ACTION SAW_active:
(*
Copyright (c) 2019 Manuel Goester, Michael Witt, Klaus Kammerer
Institute of Databases and Information Systems, Ulm University, Germany

Permission is hereby granted, free of charge, to any person obtaining a copy 
of this software and associated documentation files (the "Software"), to deal 
in the Software without restriction, including without limitation the rights 
to use, copy, modify, merge, publish, distribute, sublicense, and/or sell 
copies of the Software, and to permit persons to whom the Software is 
furnished to do so, subject to the following conditions:

The above copyright notice and this permission notice shall be included in 
all copies or substantial portions of the Software.

THE SOFTWARE IS PROVIDED "AS IS", WITHOUT WARRANTY OF ANY KIND, EXPRESS OR 
IMPLIED, INCLUDING BUT NOT LIMITED TO THE WARRANTIES OF MERCHANTABILITY, 
FITNESS FOR A PARTICULAR PURPOSE AND NONINFRINGEMENT. IN NO EVENT SHALL THE 
AUTHORS OR COPYRIGHT HOLDERS BE LIABLE FOR ANY CLAIM, DAMAGES OR OTHER 
LIABILITY, WHETHER IN AN ACTION OF CONTRACT, TORT OR OTHERWISE, ARISING FROM, 
OUT OF OR IN CONNECTION WITH THE SOFTWARE OR THE USE OR OTHER DEALINGS 
IN THE SOFTWARE.
*)
CASE stepSaw OF
	1:	
		IF FUR.currWSaw.state <> W_State.NULL THEN
			IF FUR.currWSaw.format.sawEnabled THEN
				// bring w to saw
				//SM.currW.state := StateEnum.AT_FUR_AT_SAW;
				IF NOT(FUR.sRaPosSaw) THEN
					FUR.mRaClockwise := TRUE;
				ELSE
					FUR.mRaClockwise := FALSE;
					stepSaw := stepSaw + 1;
				END_IF
			ELSE
				// skip saw and bring w directly to SL
				stepSaw := stepSaw + 2;
			END_IF
		END_IF
	2:
		// saw
		timer(IN:= TRUE, PT := FUR.currWSaw.format.sawDuration);
		FUR.mSaw := TRUE;
		IF NOT(timer.Q = FALSE AND timer.IN) THEN
			timer(IN:=FALSE);
			FUR.mSaw := FALSE;
			//FUR.state := FUR_State.FUR_SAW_FINISHED;
			stepSaw := stepSaw + 1;
		END_IF
	3: 
		IF SL.currW.state = W_State.NULL THEN
			// bring w to SL
			// SM.currW.state := StateEnum.AT_FUR_ON_CONVEYOR;
			// bend pointers of SL to current workpiece
			SL.bIdx := FUR.bIdxSaw;
			SL.wIdx := FUR.wIdxSaw;
			SL.currW := TC.batchJobQueue.batchJobs[SL.bIdx].workpieces[SL.wIdx];
			// reset own pointers
			FUR.bIdxSaw := 0;
			FUR.wIdxSaw := 0;
			FUR.currWSaw := TC.nullW;
			
			stepSaw := stepSaw + 1;
		ELSE
			// wait for SL to be ready to take a new w
		END_IF
		
	4:
		// bring w to SL
		IF NOT(FUR.sRaPosConveyorBelt) THEN
			FUR.mRaClockwise := TRUE;
		ELSE
			FUR.mRaClockwise := FALSE;
			FUR.compressor := TRUE;
			FUR.valveSlider := TRUE;
		END_IF
		
		IF SL.lbEntry THEN
			FUR.mConveyorBeltForward := TRUE;
		ELSE
			FUR.mConveyorBeltForward := FALSE;
			FUR.compressor := FALSE;
			FUR.valveSlider := FALSE;
			//FUR.state := FUR_State.FUR_W_FINISHED_BACK_TO_DEFAULT;
			stepSaw := stepSaw + 1;
		END_IF
	5:
		// get rotating desk back to succer pos
		IF NOT(FUR.sRaPosSucker) THEN
			FUR.mRaCClockwise := TRUE;
		ELSE
			FUR.mRaCClockwise := FALSE;
			// finsihed, go back to 1 to wait for next w
			stepSaw := 1;
		END_IF
END_CASE
END_ACTION

ACTION TO_DEFAULT_POS_active:
(*
Copyright (c) 2019 Manuel Goester, Michael Witt, Klaus Kammerer
Institute of Databases and Information Systems, Ulm University, Germany

Permission is hereby granted, free of charge, to any person obtaining a copy 
of this software and associated documentation files (the "Software"), to deal 
in the Software without restriction, including without limitation the rights 
to use, copy, modify, merge, publish, distribute, sublicense, and/or sell 
copies of the Software, and to permit persons to whom the Software is 
furnished to do so, subject to the following conditions:

The above copyright notice and this permission notice shall be included in 
all copies or substantial portions of the Software.

THE SOFTWARE IS PROVIDED "AS IS", WITHOUT WARRANTY OF ANY KIND, EXPRESS OR 
IMPLIED, INCLUDING BUT NOT LIMITED TO THE WARRANTIES OF MERCHANTABILITY, 
FITNESS FOR A PARTICULAR PURPOSE AND NONINFRINGEMENT. IN NO EVENT SHALL THE 
AUTHORS OR COPYRIGHT HOLDERS BE LIABLE FOR ANY CLAIM, DAMAGES OR OTHER 
LIABILITY, WHETHER IN AN ACTION OF CONTRACT, TORT OR OTHERWISE, ARISING FROM, 
OUT OF OR IN CONNECTION WITH THE SOFTWARE OR THE USE OR OTHER DEALINGS 
IN THE SOFTWARE.
*)
IF NOT(FUR.sFurnanceSliderOutside) THEN
	FUR.mFurnanceSliderOut := TRUE;
	FUR.compressor := TRUE;
	FUR.valveFurnanceDoor := TRUE;
ELSE
	FUR.mFurnanceSliderOut := FALSE;
	FUR.compressor := FALSE;
	FUR.valveFurnanceDoor := FALSE;
END_IF

IF NOT(FUR.sSuckerPosRa) THEN
	FUR.mSuckertoRa := TRUE;
ELSE
	FUR.mSuckertoRa := FALSE;
END_IF

IF NOT(FUR.sRaPosSucker) THEN
	FUR.mRaCClockwise := TRUE;
ELSE
	FUR.mRaCClockwise := FALSE;
END_IF

IF FUR.sSuckerPosRa AND FUR.sRaPosSucker AND FUR.sFurnanceSliderOutside THEN
	fin := TRUE;
END_IF
END_ACTION

ACTION TO_DEFAULT_POS_exit:
(*
Copyright (c) 2019 Manuel Goester, Michael Witt, Klaus Kammerer
Institute of Databases and Information Systems, Ulm University, Germany

Permission is hereby granted, free of charge, to any person obtaining a copy 
of this software and associated documentation files (the "Software"), to deal 
in the Software without restriction, including without limitation the rights 
to use, copy, modify, merge, publish, distribute, sublicense, and/or sell 
copies of the Software, and to permit persons to whom the Software is 
furnished to do so, subject to the following conditions:

The above copyright notice and this permission notice shall be included in 
all copies or substantial portions of the Software.

THE SOFTWARE IS PROVIDED "AS IS", WITHOUT WARRANTY OF ANY KIND, EXPRESS OR 
IMPLIED, INCLUDING BUT NOT LIMITED TO THE WARRANTIES OF MERCHANTABILITY, 
FITNESS FOR A PARTICULAR PURPOSE AND NONINFRINGEMENT. IN NO EVENT SHALL THE 
AUTHORS OR COPYRIGHT HOLDERS BE LIABLE FOR ANY CLAIM, DAMAGES OR OTHER 
LIABILITY, WHETHER IN AN ACTION OF CONTRACT, TORT OR OTHERWISE, ARISING FROM, 
OUT OF OR IN CONNECTION WITH THE SOFTWARE OR THE USE OR OTHER DEALINGS 
IN THE SOFTWARE.
*)
fin := FALSE;
END_ACTION

END_PROGRAM

// Device/Application/FUR/FBs/FUR_BURN
(*
	Function Block for buring a workpiece in furnace
	w : Workpiece to be burned

Copyright (c) 2019 Manuel Goester, Michael Witt, Klaus Kammerer
Institute of Databases and Information Systems, Ulm University, Germany

Permission is hereby granted, free of charge, to any person obtaining a copy 
of this software and associated documentation files (the "Software"), to deal 
in the Software without restriction, including without limitation the rights 
to use, copy, modify, merge, publish, distribute, sublicense, and/or sell 
copies of the Software, and to permit persons to whom the Software is 
furnished to do so, subject to the following conditions:

The above copyright notice and this permission notice shall be included in 
all copies or substantial portions of the Software.

THE SOFTWARE IS PROVIDED "AS IS", WITHOUT WARRANTY OF ANY KIND, EXPRESS OR 
IMPLIED, INCLUDING BUT NOT LIMITED TO THE WARRANTIES OF MERCHANTABILITY, 
FITNESS FOR A PARTICULAR PURPOSE AND NONINFRINGEMENT. IN NO EVENT SHALL THE 
AUTHORS OR COPYRIGHT HOLDERS BE LIABLE FOR ANY CLAIM, DAMAGES OR OTHER 
LIABILITY, WHETHER IN AN ACTION OF CONTRACT, TORT OR OTHERWISE, ARISING FROM, 
OUT OF OR IN CONNECTION WITH THE SOFTWARE OR THE USE OR OTHER DEALINGS 
IN THE SOFTWARE.
*)
FUNCTION_BLOCK FUR_BURN
VAR_INPUT
	w: Workpiece;
END_VAR
VAR_OUTPUT
END_VAR
VAR
	step: INT := 1;
	fin: BOOL := FALSE;
	stepFin: BOOL := FALSE;
	timer: TON;
END_VAR

CASE step OF
	1:	// open door and drive workpiece into furnace
		// reset flag
		fin := FALSE;
		FUR.compressor := TRUE;
		FUR.valveFurnanceDoor := TRUE;
		IF FUR.sFurnanceSliderInside = FALSE THEN
			FUR.mFurnanceSliderIn := TRUE;
		ELSE
			FUR.mFurnanceSliderIn := FALSE;
			FUR.state := FUR_State.FUR_WAGON_INSIDE;
			step := step + 1;
		END_IF
	2:	// burn
		IF FUR.state = FUR_State.FUR_WAGON_INSIDE THEN
			//SM.currW.state := StateEnum.AT_FUR_IN_FUR;
			timer(IN:= TRUE, PT := FUR.currWBurner.format.furDuration);
			FUR.valveFurnanceDoor := FALSE;
			IF NOT(timer.Q = FALSE AND timer.IN) THEN
				// reset timer
				timer(IN:= FALSE);
				FUR.compressor := TRUE;
				FUR.valveFurnanceDoor := TRUE;
				FUR.state := FUR_State.FUR_BURNED;
				step := step + 1;
			END_IF
		END_IF
	3:	// drive slider out
		IF FUR.state = FUR_State.FUR_BURNED THEN
			//SM.currW.state := StateEnum.AT_FUR_IN_WAGON;
			IF FUR.sFurnanceSliderOutside = FALSE THEN
				FUR.mFurnanceSliderOut := TRUE;
			ELSE
				FUR.mFurnanceSliderOut := FALSE;
				FUR.state := FUR_State.FUR_WAGON_OUTSIDE;
				FUR.compressor := FALSE;
				FUR.valveFurnanceDoor := FALSE;
				step := step + 1;
			END_IF
		END_IF
	4:	// finished
		fin := TRUE;
		step := 1;
END_CASE

END_FUNCTION_BLOCK

// Device/Application/VG/VG_SINGLE_MODE
PROGRAM VG_SINGLE_MODE
VAR
	vg_move: VG_MOVE;
	vg_move_to_pos: VG_MOVE_TO_POS;
	xFin: BOOL;
	yFin: BOOL;
	zFin: BOOL;
	pneumatic_loaded: BOOL;
	timer: TON;
	subBlockStart: BOOL;
	fin: BOOL;
	step: INT := 1;
END_VAR

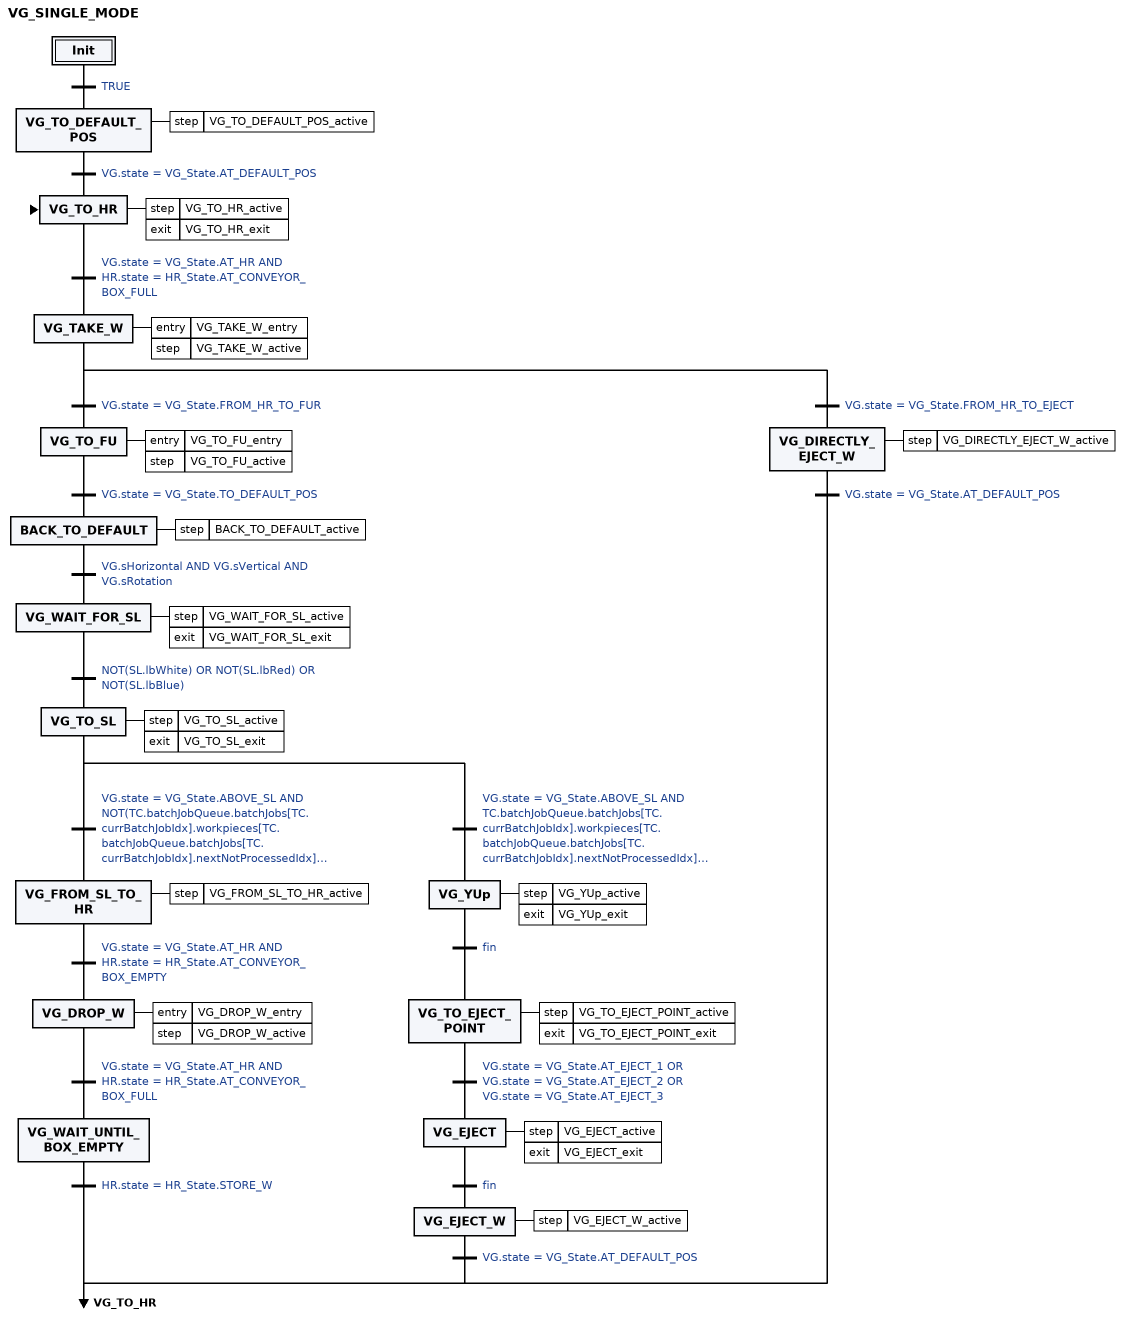
INITIAL_STEP Init:
END_STEP
TRANSITION FROM Init TO VG_TO_DEFAULT_POS
    := TRUE;
END_TRANSITION
STEP VG_TO_DEFAULT_POS:
    VG_TO_DEFAULT_POS_active(N);  // step action
END_STEP
TRANSITION FROM VG_TO_DEFAULT_POS TO VG_TO_HR
    := VG.state = VG_State.AT_DEFAULT_POS;
END_TRANSITION
STEP VG_TO_HR:
    VG_TO_HR_active(N);  // step action
    VG_TO_HR_exit(P0);  // exit action
END_STEP
TRANSITION FROM VG_TO_HR TO VG_TAKE_W
    := VG.state = VG_State.AT_HR AND HR.state = HR_State.AT_CONVEYOR_BOX_FULL;
END_TRANSITION
STEP VG_TAKE_W:
    VG_TAKE_W_entry(P1);  // entry action
    VG_TAKE_W_active(N);  // step action
END_STEP
TRANSITION FROM VG_TAKE_W TO VG_TO_FU
    := VG.state = VG_State.FROM_HR_TO_FUR;
END_TRANSITION
STEP VG_TO_FU:
    VG_TO_FU_entry(P1);  // entry action
    VG_TO_FU_active(N);  // step action
END_STEP
TRANSITION FROM VG_TO_FU TO BACK_TO_DEFAULT
    := VG.state = VG_State.TO_DEFAULT_POS;
END_TRANSITION
STEP BACK_TO_DEFAULT:
    BACK_TO_DEFAULT_active(N);  // step action
END_STEP
TRANSITION FROM BACK_TO_DEFAULT TO VG_WAIT_FOR_SL
    := VG.sHorizontal AND VG.sVertical AND VG.sRotation;
END_TRANSITION
STEP VG_WAIT_FOR_SL:
    VG_WAIT_FOR_SL_active(N);  // step action
    VG_WAIT_FOR_SL_exit(P0);  // exit action
END_STEP
TRANSITION FROM VG_WAIT_FOR_SL TO VG_TO_SL
    := NOT(SL.lbWhite) OR NOT(SL.lbRed) OR NOT(SL.lbBlue);
END_TRANSITION
STEP VG_TO_SL:
    VG_TO_SL_active(N);  // step action
    VG_TO_SL_exit(P0);  // exit action
END_STEP
TRANSITION FROM VG_TO_SL TO VG_FROM_SL_TO_HR
    := VG.state = VG_State.ABOVE_SL AND NOT(TC.batchJobQueue.batchJobs[TC.currBatchJobIdx].workpieces[TC.batchJobQueue.batchJobs[TC.currBatchJobIdx].nextNotProcessedIdx].format.ejectEnabled);
END_TRANSITION
STEP VG_FROM_SL_TO_HR:
    VG_FROM_SL_TO_HR_active(N);  // step action
END_STEP
TRANSITION FROM VG_FROM_SL_TO_HR TO VG_DROP_W
    := VG.state = VG_State.AT_HR AND HR.state = HR_State.AT_CONVEYOR_BOX_EMPTY;
END_TRANSITION
STEP VG_DROP_W:
    VG_DROP_W_entry(P1);  // entry action
    VG_DROP_W_active(N);  // step action
END_STEP
TRANSITION FROM VG_DROP_W TO VG_WAIT_UNTIL_BOX_EMPTY
    := VG.state = VG_State.AT_HR AND HR.state = HR_State.AT_CONVEYOR_BOX_FULL;
END_TRANSITION
STEP VG_WAIT_UNTIL_BOX_EMPTY:
END_STEP
TRANSITION FROM VG_WAIT_UNTIL_BOX_EMPTY TO VG_TO_HR
    := HR.state = HR_State.STORE_W;
END_TRANSITION
TRANSITION FROM VG_TO_SL TO VG_YUp
    := VG.state = VG_State.ABOVE_SL AND TC.batchJobQueue.batchJobs[TC.currBatchJobIdx].workpieces[TC.batchJobQueue.batchJobs[TC.currBatchJobIdx].nextNotProcessedIdx].format.ejectEnabled;
END_TRANSITION
STEP VG_YUp:
    VG_YUp_active(N);  // step action
    VG_YUp_exit(P0);  // exit action
END_STEP
TRANSITION FROM VG_YUp TO VG_TO_EJECT_POINT
    := fin;
END_TRANSITION
STEP VG_TO_EJECT_POINT:
    VG_TO_EJECT_POINT_active(N);  // step action
    VG_TO_EJECT_POINT_exit(P0);  // exit action
END_STEP
TRANSITION FROM VG_TO_EJECT_POINT TO VG_EJECT
    := VG.state = VG_State.AT_EJECT_1 OR VG.state = VG_State.AT_EJECT_2 OR VG.state = VG_State.AT_EJECT_3;
END_TRANSITION
STEP VG_EJECT:
    VG_EJECT_active(N);  // step action
    VG_EJECT_exit(P0);  // exit action
END_STEP
TRANSITION FROM VG_EJECT TO VG_EJECT_W
    := fin;
END_TRANSITION
STEP VG_EJECT_W:
    VG_EJECT_W_active(N);  // step action
END_STEP
TRANSITION FROM VG_EJECT_W TO VG_TO_HR
    := VG.state = VG_State.AT_DEFAULT_POS;
END_TRANSITION
TRANSITION FROM VG_TAKE_W TO VG_DIRECTLY_EJECT_W
    := VG.state = VG_State.FROM_HR_TO_EJECT;
END_TRANSITION
STEP VG_DIRECTLY_EJECT_W:
    VG_DIRECTLY_EJECT_W_active(N);  // step action
END_STEP
TRANSITION FROM VG_DIRECTLY_EJECT_W TO VG_TO_HR
    := VG.state = VG_State.AT_DEFAULT_POS;
END_TRANSITION

ACTION XForward_VG_TAKE_W_active_exit:
(*
Copyright (c) 2019 Manuel Goester, Michael Witt, Klaus Kammerer
Institute of Databases and Information Systems, Ulm University, Germany

Permission is hereby granted, free of charge, to any person obtaining a copy 
of this software and associated documentation files (the "Software"), to deal 
in the Software without restriction, including without limitation the rights 
to use, copy, modify, merge, publish, distribute, sublicense, and/or sell 
copies of the Software, and to permit persons to whom the Software is 
furnished to do so, subject to the following conditions:

The above copyright notice and this permission notice shall be included in 
all copies or substantial portions of the Software.

THE SOFTWARE IS PROVIDED "AS IS", WITHOUT WARRANTY OF ANY KIND, EXPRESS OR 
IMPLIED, INCLUDING BUT NOT LIMITED TO THE WARRANTIES OF MERCHANTABILITY, 
FITNESS FOR A PARTICULAR PURPOSE AND NONINFRINGEMENT. IN NO EVENT SHALL THE 
AUTHORS OR COPYRIGHT HOLDERS BE LIABLE FOR ANY CLAIM, DAMAGES OR OTHER 
LIABILITY, WHETHER IN AN ACTION OF CONTRACT, TORT OR OTHERWISE, ARISING FROM, 
OUT OF OR IN CONNECTION WITH THE SOFTWARE OR THE USE OR OTHER DEALINGS 
IN THE SOFTWARE.
*)
xFin := FALSE;
END_ACTION

ACTION YUp_VG_DROP_W_active_exit:
(*
Copyright (c) 2019 Manuel Goester, Michael Witt, Klaus Kammerer
Institute of Databases and Information Systems, Ulm University, Germany

Permission is hereby granted, free of charge, to any person obtaining a copy 
of this software and associated documentation files (the "Software"), to deal 
in the Software without restriction, including without limitation the rights 
to use, copy, modify, merge, publish, distribute, sublicense, and/or sell 
copies of the Software, and to permit persons to whom the Software is 
furnished to do so, subject to the following conditions:

The above copyright notice and this permission notice shall be included in 
all copies or substantial portions of the Software.

THE SOFTWARE IS PROVIDED "AS IS", WITHOUT WARRANTY OF ANY KIND, EXPRESS OR 
IMPLIED, INCLUDING BUT NOT LIMITED TO THE WARRANTIES OF MERCHANTABILITY, 
FITNESS FOR A PARTICULAR PURPOSE AND NONINFRINGEMENT. IN NO EVENT SHALL THE 
AUTHORS OR COPYRIGHT HOLDERS BE LIABLE FOR ANY CLAIM, DAMAGES OR OTHER 
LIABILITY, WHETHER IN AN ACTION OF CONTRACT, TORT OR OTHERWISE, ARISING FROM, 
OUT OF OR IN CONNECTION WITH THE SOFTWARE OR THE USE OR OTHER DEALINGS 
IN THE SOFTWARE.
*)
yFin := FALSE;
VG.state := VG_State.AT_HR;
VG_SINGLE_MODE.subBlockStart := FALSE;
END_ACTION

ACTION VG_TO_FU_entry:
(*
Copyright (c) 2019 Manuel Goester, Michael Witt, Klaus Kammerer
Institute of Databases and Information Systems, Ulm University, Germany

Permission is hereby granted, free of charge, to any person obtaining a copy 
of this software and associated documentation files (the "Software"), to deal 
in the Software without restriction, including without limitation the rights 
to use, copy, modify, merge, publish, distribute, sublicense, and/or sell 
copies of the Software, and to permit persons to whom the Software is 
furnished to do so, subject to the following conditions:

The above copyright notice and this permission notice shall be included in 
all copies or substantial portions of the Software.

THE SOFTWARE IS PROVIDED "AS IS", WITHOUT WARRANTY OF ANY KIND, EXPRESS OR 
IMPLIED, INCLUDING BUT NOT LIMITED TO THE WARRANTIES OF MERCHANTABILITY, 
FITNESS FOR A PARTICULAR PURPOSE AND NONINFRINGEMENT. IN NO EVENT SHALL THE 
AUTHORS OR COPYRIGHT HOLDERS BE LIABLE FOR ANY CLAIM, DAMAGES OR OTHER 
LIABILITY, WHETHER IN AN ACTION OF CONTRACT, TORT OR OTHERWISE, ARISING FROM, 
OUT OF OR IN CONNECTION WITH THE SOFTWARE OR THE USE OR OTHER DEALINGS 
IN THE SOFTWARE.
*)
VG_SINGLE_MODE.subBlockStart := TRUE;
END_ACTION

ACTION ZBack_VG_FROM_SL_TO_HR_active_exit:
(*
Copyright (c) 2019 Manuel Goester, Michael Witt, Klaus Kammerer
Institute of Databases and Information Systems, Ulm University, Germany

Permission is hereby granted, free of charge, to any person obtaining a copy 
of this software and associated documentation files (the "Software"), to deal 
in the Software without restriction, including without limitation the rights 
to use, copy, modify, merge, publish, distribute, sublicense, and/or sell 
copies of the Software, and to permit persons to whom the Software is 
furnished to do so, subject to the following conditions:

The above copyright notice and this permission notice shall be included in 
all copies or substantial portions of the Software.

THE SOFTWARE IS PROVIDED "AS IS", WITHOUT WARRANTY OF ANY KIND, EXPRESS OR 
IMPLIED, INCLUDING BUT NOT LIMITED TO THE WARRANTIES OF MERCHANTABILITY, 
FITNESS FOR A PARTICULAR PURPOSE AND NONINFRINGEMENT. IN NO EVENT SHALL THE 
AUTHORS OR COPYRIGHT HOLDERS BE LIABLE FOR ANY CLAIM, DAMAGES OR OTHER 
LIABILITY, WHETHER IN AN ACTION OF CONTRACT, TORT OR OTHERWISE, ARISING FROM, 
OUT OF OR IN CONNECTION WITH THE SOFTWARE OR THE USE OR OTHER DEALINGS 
IN THE SOFTWARE.
*)
zFin := FALSE;
END_ACTION

ACTION Suction_VG_TAKE_W_active_active:
(*
Copyright (c) 2019 Manuel Goester, Michael Witt, Klaus Kammerer
Institute of Databases and Information Systems, Ulm University, Germany

Permission is hereby granted, free of charge, to any person obtaining a copy 
of this software and associated documentation files (the "Software"), to deal 
in the Software without restriction, including without limitation the rights 
to use, copy, modify, merge, publish, distribute, sublicense, and/or sell 
copies of the Software, and to permit persons to whom the Software is 
furnished to do so, subject to the following conditions:

The above copyright notice and this permission notice shall be included in 
all copies or substantial portions of the Software.

THE SOFTWARE IS PROVIDED "AS IS", WITHOUT WARRANTY OF ANY KIND, EXPRESS OR 
IMPLIED, INCLUDING BUT NOT LIMITED TO THE WARRANTIES OF MERCHANTABILITY, 
FITNESS FOR A PARTICULAR PURPOSE AND NONINFRINGEMENT. IN NO EVENT SHALL THE 
AUTHORS OR COPYRIGHT HOLDERS BE LIABLE FOR ANY CLAIM, DAMAGES OR OTHER 
LIABILITY, WHETHER IN AN ACTION OF CONTRACT, TORT OR OTHERWISE, ARISING FROM, 
OUT OF OR IN CONNECTION WITH THE SOFTWARE OR THE USE OR OTHER DEALINGS 
IN THE SOFTWARE.
*)
IF pneumatic_loaded = FALSE THEN
	VG.valve := TRUE;
	// init timer
	timer(IN:= TRUE, PT:= T#2S);
	
	IF timer.Q = FALSE AND timer.IN THEN
		// go
		VG.compressor := TRUE;
	ELSE
		// stop
		VG.compressor := FALSE;
		
		// reset timer
		timer(IN:= FALSE);
		
		// go to next step
		pneumatic_loaded := TRUE;
	END_IF
ELSE
	// reset timer
	timer(IN:= FALSE);
END_IF
END_ACTION

ACTION ZBack_VG_TO_FU_active_active:
(*
Copyright (c) 2019 Manuel Goester, Michael Witt, Klaus Kammerer
Institute of Databases and Information Systems, Ulm University, Germany

Permission is hereby granted, free of charge, to any person obtaining a copy 
of this software and associated documentation files (the "Software"), to deal 
in the Software without restriction, including without limitation the rights 
to use, copy, modify, merge, publish, distribute, sublicense, and/or sell 
copies of the Software, and to permit persons to whom the Software is 
furnished to do so, subject to the following conditions:

The above copyright notice and this permission notice shall be included in 
all copies or substantial portions of the Software.

THE SOFTWARE IS PROVIDED "AS IS", WITHOUT WARRANTY OF ANY KIND, EXPRESS OR 
IMPLIED, INCLUDING BUT NOT LIMITED TO THE WARRANTIES OF MERCHANTABILITY, 
FITNESS FOR A PARTICULAR PURPOSE AND NONINFRINGEMENT. IN NO EVENT SHALL THE 
AUTHORS OR COPYRIGHT HOLDERS BE LIABLE FOR ANY CLAIM, DAMAGES OR OTHER 
LIABILITY, WHETHER IN AN ACTION OF CONTRACT, TORT OR OTHERWISE, ARISING FROM, 
OUT OF OR IN CONNECTION WITH THE SOFTWARE OR THE USE OR OTHER DEALINGS 
IN THE SOFTWARE.
*)
IF NOT(VG.sHorizontal) THEN
	VG.mHorizontalBackward := TRUE;
ELSE
	VG.mHorizontalBackward := FALSE;
	zFin := TRUE;
END_IF
END_ACTION

ACTION VG_TO_SL_active:
(*
Copyright (c) 2019 Manuel Goester, Michael Witt, Klaus Kammerer
Institute of Databases and Information Systems, Ulm University, Germany

Permission is hereby granted, free of charge, to any person obtaining a copy 
of this software and associated documentation files (the "Software"), to deal 
in the Software without restriction, including without limitation the rights 
to use, copy, modify, merge, publish, distribute, sublicense, and/or sell 
copies of the Software, and to permit persons to whom the Software is 
furnished to do so, subject to the following conditions:

The above copyright notice and this permission notice shall be included in 
all copies or substantial portions of the Software.

THE SOFTWARE IS PROVIDED "AS IS", WITHOUT WARRANTY OF ANY KIND, EXPRESS OR 
IMPLIED, INCLUDING BUT NOT LIMITED TO THE WARRANTIES OF MERCHANTABILITY, 
FITNESS FOR A PARTICULAR PURPOSE AND NONINFRINGEMENT. IN NO EVENT SHALL THE 
AUTHORS OR COPYRIGHT HOLDERS BE LIABLE FOR ANY CLAIM, DAMAGES OR OTHER 
LIABILITY, WHETHER IN AN ACTION OF CONTRACT, TORT OR OTHERWISE, ARISING FROM, 
OUT OF OR IN CONNECTION WITH THE SOFTWARE OR THE USE OR OTHER DEALINGS 
IN THE SOFTWARE.
*)
CASE step OF
	1:
		// decide to which positon of SL VG will go
		IF NOT(SL.lbWhite) THEN
			// go to sorting line pos 1: 
			VG.state := VG_State.TO_SL_OUTPUT_1;
			step := step + 1;
		ELSIF NOT(SL.lbRed) THEN
			// go to sorting line pos 2: 
			VG.state := VG_State.TO_SL_OUTPUT_2;
			step := step + 1;
		ELSIF NOT(SL.lbBlue) THEN
			// go to sorting line pos 3: 
			VG.state := VG_State.TO_SL_OUTPUT_3;
			step := step + 1;
		END_IF
	2:
		// x and z axis: move to SL 
		IF NOT(fin) THEN
			CASE VG.state OF
				VG_State.TO_SL_OUTPUT_1:
					vg_move_to_pos(x := 58, y := 0, z := 69);
				VG_State.TO_SL_OUTPUT_2:
					vg_move_to_pos(x := 63, y := 0, z := 57);
				VG_State.TO_SL_OUTPUT_3:
					vg_move_to_pos(x := 87, y := 0, z := 47);
			END_CASE
			fin := vg_move_to_pos.fin;
		ELSE
			fin := FALSE;
			step := step + 1;
		END_IF
	3:
		// y axis: move to SL
		IF NOT(fin) THEN
			CASE VG.state OF
				VG_State.TO_SL_OUTPUT_1:
					vg_move_to_pos(x := 58, y := 125, z := 69);
					TC.batchJobQueue.batchJobs[TC.currBatchJobIdx].workpieces[TC.batchJobQueue.batchJobs[TC.currBatchJobIdx].nextNotProcessedIdx].sortingLinePos := 1;
				VG_State.TO_SL_OUTPUT_2:
					vg_move_to_pos(x := 63, y := 125, z := 57);
					TC.batchJobQueue.batchJobs[TC.currBatchJobIdx].workpieces[TC.batchJobQueue.batchJobs[TC.currBatchJobIdx].nextNotProcessedIdx].sortingLinePos := 2;
				VG_State.TO_SL_OUTPUT_3:
					vg_move_to_pos(x := 87, y := 125, z := 47);
					TC.batchJobQueue.batchJobs[TC.currBatchJobIdx].workpieces[TC.batchJobQueue.batchJobs[TC.currBatchJobIdx].nextNotProcessedIdx].sortingLinePos := 3;
			END_CASE
			fin := vg_move_to_pos.fin;
		ELSE
			fin := FALSE;
			step := step + 1;
		END_IF
	4:
		CASE VG.state OF
			VG_State.TO_SL_OUTPUT_1:
				VG.state := VG_State.AT_SL_OUTPUT_1;
			VG_State.TO_SL_OUTPUT_2:
				VG.state := VG_State.AT_SL_OUTPUT_2;
			VG_State.TO_SL_OUTPUT_3:
				VG.state := VG_State.AT_SL_OUTPUT_3;
		END_CASE
		// succ workpiece
		IF pneumatic_loaded = FALSE THEN
			VG.valve := TRUE;
			// init timer
			timer(IN:= TRUE, PT:= T#2S);
			IF timer.Q = FALSE AND timer.IN THEN
				// go
				VG.compressor := TRUE;
			ELSE
				// stop
				VG.compressor := FALSE;
				// reset timer
				timer(IN:= FALSE);
				// set flag
				pneumatic_loaded := TRUE;
			END_IF
		ELSE
			step := step + 1;
		END_IF
	5:
		// y axis: move up
		IF NOT(VG.sVertical) THEN
			VG.mVerticalUp := TRUE;
		ELSE
			VG.mVerticalUp := FALSE;
			VG.cY := 0;
			step := step + 1;
		END_IF
	6:
		// finsihed
		VG.state := VG_State.ABOVE_SL;
END_CASE
END_ACTION

ACTION YDown_VG_TO_FU_active_exit:
(*
Copyright (c) 2019 Manuel Goester, Michael Witt, Klaus Kammerer
Institute of Databases and Information Systems, Ulm University, Germany

Permission is hereby granted, free of charge, to any person obtaining a copy 
of this software and associated documentation files (the "Software"), to deal 
in the Software without restriction, including without limitation the rights 
to use, copy, modify, merge, publish, distribute, sublicense, and/or sell 
copies of the Software, and to permit persons to whom the Software is 
furnished to do so, subject to the following conditions:

The above copyright notice and this permission notice shall be included in 
all copies or substantial portions of the Software.

THE SOFTWARE IS PROVIDED "AS IS", WITHOUT WARRANTY OF ANY KIND, EXPRESS OR 
IMPLIED, INCLUDING BUT NOT LIMITED TO THE WARRANTIES OF MERCHANTABILITY, 
FITNESS FOR A PARTICULAR PURPOSE AND NONINFRINGEMENT. IN NO EVENT SHALL THE 
AUTHORS OR COPYRIGHT HOLDERS BE LIABLE FOR ANY CLAIM, DAMAGES OR OTHER 
LIABILITY, WHETHER IN AN ACTION OF CONTRACT, TORT OR OTHERWISE, ARISING FROM, 
OUT OF OR IN CONNECTION WITH THE SOFTWARE OR THE USE OR OTHER DEALINGS 
IN THE SOFTWARE.
*)
fin := FALSE;
END_ACTION

ACTION ZBack_VG_TO_FU_active_exit_0:
(*
Copyright (c) 2019 Manuel Goester, Michael Witt, Klaus Kammerer
Institute of Databases and Information Systems, Ulm University, Germany

Permission is hereby granted, free of charge, to any person obtaining a copy 
of this software and associated documentation files (the "Software"), to deal 
in the Software without restriction, including without limitation the rights 
to use, copy, modify, merge, publish, distribute, sublicense, and/or sell 
copies of the Software, and to permit persons to whom the Software is 
furnished to do so, subject to the following conditions:

The above copyright notice and this permission notice shall be included in 
all copies or substantial portions of the Software.

THE SOFTWARE IS PROVIDED "AS IS", WITHOUT WARRANTY OF ANY KIND, EXPRESS OR 
IMPLIED, INCLUDING BUT NOT LIMITED TO THE WARRANTIES OF MERCHANTABILITY, 
FITNESS FOR A PARTICULAR PURPOSE AND NONINFRINGEMENT. IN NO EVENT SHALL THE 
AUTHORS OR COPYRIGHT HOLDERS BE LIABLE FOR ANY CLAIM, DAMAGES OR OTHER 
LIABILITY, WHETHER IN AN ACTION OF CONTRACT, TORT OR OTHERWISE, ARISING FROM, 
OUT OF OR IN CONNECTION WITH THE SOFTWARE OR THE USE OR OTHER DEALINGS 
IN THE SOFTWARE.
*)
zFin := FALSE;
END_ACTION

ACTION Wait_VG_DROP_W_active_active:
(*
Copyright (c) 2019 Manuel Goester, Michael Witt, Klaus Kammerer
Institute of Databases and Information Systems, Ulm University, Germany

Permission is hereby granted, free of charge, to any person obtaining a copy 
of this software and associated documentation files (the "Software"), to deal 
in the Software without restriction, including without limitation the rights 
to use, copy, modify, merge, publish, distribute, sublicense, and/or sell 
copies of the Software, and to permit persons to whom the Software is 
furnished to do so, subject to the following conditions:

The above copyright notice and this permission notice shall be included in 
all copies or substantial portions of the Software.

THE SOFTWARE IS PROVIDED "AS IS", WITHOUT WARRANTY OF ANY KIND, EXPRESS OR 
IMPLIED, INCLUDING BUT NOT LIMITED TO THE WARRANTIES OF MERCHANTABILITY, 
FITNESS FOR A PARTICULAR PURPOSE AND NONINFRINGEMENT. IN NO EVENT SHALL THE 
AUTHORS OR COPYRIGHT HOLDERS BE LIABLE FOR ANY CLAIM, DAMAGES OR OTHER 
LIABILITY, WHETHER IN AN ACTION OF CONTRACT, TORT OR OTHERWISE, ARISING FROM, 
OUT OF OR IN CONNECTION WITH THE SOFTWARE OR THE USE OR OTHER DEALINGS 
IN THE SOFTWARE.
*)
timer(IN:= TRUE, PT:= T#1S);
IF NOT(timer.Q = FALSE AND timer.IN) THEN
	// reset timer
	timer(IN:= FALSE);
	// go to next step
	fin := TRUE;
END_IF
END_ACTION

ACTION XForward_VG_TAKE_W_active_active:
(*
Copyright (c) 2019 Manuel Goester, Michael Witt, Klaus Kammerer
Institute of Databases and Information Systems, Ulm University, Germany

Permission is hereby granted, free of charge, to any person obtaining a copy 
of this software and associated documentation files (the "Software"), to deal 
in the Software without restriction, including without limitation the rights 
to use, copy, modify, merge, publish, distribute, sublicense, and/or sell 
copies of the Software, and to permit persons to whom the Software is 
furnished to do so, subject to the following conditions:

The above copyright notice and this permission notice shall be included in 
all copies or substantial portions of the Software.

THE SOFTWARE IS PROVIDED "AS IS", WITHOUT WARRANTY OF ANY KIND, EXPRESS OR 
IMPLIED, INCLUDING BUT NOT LIMITED TO THE WARRANTIES OF MERCHANTABILITY, 
FITNESS FOR A PARTICULAR PURPOSE AND NONINFRINGEMENT. IN NO EVENT SHALL THE 
AUTHORS OR COPYRIGHT HOLDERS BE LIABLE FOR ANY CLAIM, DAMAGES OR OTHER 
LIABILITY, WHETHER IN AN ACTION OF CONTRACT, TORT OR OTHERWISE, ARISING FROM, 
OUT OF OR IN CONNECTION WITH THE SOFTWARE OR THE USE OR OTHER DEALINGS 
IN THE SOFTWARE.
*)
VG.state := VG_State.GET_W_FROM_HR;
IF NOT(xFin) THEN
	vg_move_to_pos(x:=27, y:=0, z:=206);
	xFin := vg_move_to_pos.fin;
END_IF
END_ACTION

ACTION Wait_VG_TO_FU_active_exit:
(*
Copyright (c) 2019 Manuel Goester, Michael Witt, Klaus Kammerer
Institute of Databases and Information Systems, Ulm University, Germany

Permission is hereby granted, free of charge, to any person obtaining a copy 
of this software and associated documentation files (the "Software"), to deal 
in the Software without restriction, including without limitation the rights 
to use, copy, modify, merge, publish, distribute, sublicense, and/or sell 
copies of the Software, and to permit persons to whom the Software is 
furnished to do so, subject to the following conditions:

The above copyright notice and this permission notice shall be included in 
all copies or substantial portions of the Software.

THE SOFTWARE IS PROVIDED "AS IS", WITHOUT WARRANTY OF ANY KIND, EXPRESS OR 
IMPLIED, INCLUDING BUT NOT LIMITED TO THE WARRANTIES OF MERCHANTABILITY, 
FITNESS FOR A PARTICULAR PURPOSE AND NONINFRINGEMENT. IN NO EVENT SHALL THE 
AUTHORS OR COPYRIGHT HOLDERS BE LIABLE FOR ANY CLAIM, DAMAGES OR OTHER 
LIABILITY, WHETHER IN AN ACTION OF CONTRACT, TORT OR OTHERWISE, ARISING FROM, 
OUT OF OR IN CONNECTION WITH THE SOFTWARE OR THE USE OR OTHER DEALINGS 
IN THE SOFTWARE.
*)
fin := FALSE;
END_ACTION

ACTION YDown_VG_DROP_W_active_active:
(*
Copyright (c) 2019 Manuel Goester, Michael Witt, Klaus Kammerer
Institute of Databases and Information Systems, Ulm University, Germany

Permission is hereby granted, free of charge, to any person obtaining a copy 
of this software and associated documentation files (the "Software"), to deal 
in the Software without restriction, including without limitation the rights 
to use, copy, modify, merge, publish, distribute, sublicense, and/or sell 
copies of the Software, and to permit persons to whom the Software is 
furnished to do so, subject to the following conditions:

The above copyright notice and this permission notice shall be included in 
all copies or substantial portions of the Software.

THE SOFTWARE IS PROVIDED "AS IS", WITHOUT WARRANTY OF ANY KIND, EXPRESS OR 
IMPLIED, INCLUDING BUT NOT LIMITED TO THE WARRANTIES OF MERCHANTABILITY, 
FITNESS FOR A PARTICULAR PURPOSE AND NONINFRINGEMENT. IN NO EVENT SHALL THE 
AUTHORS OR COPYRIGHT HOLDERS BE LIABLE FOR ANY CLAIM, DAMAGES OR OTHER 
LIABILITY, WHETHER IN AN ACTION OF CONTRACT, TORT OR OTHERWISE, ARISING FROM, 
OUT OF OR IN CONNECTION WITH THE SOFTWARE OR THE USE OR OTHER DEALINGS 
IN THE SOFTWARE.
*)
VG.state := VG_State.DROPPING_W_TO_HR;
IF NOT(yFin) THEN
	vg_move_to_pos(x:=27, y:=45, z:=206);
	IF vg_move_to_pos.fin THEN
		yFin := TRUE;
	END_IF
END_IF
END_ACTION

ACTION VG_TO_EJECT_POINT_active:
(*
Copyright (c) 2019 Manuel Goester, Michael Witt, Klaus Kammerer
Institute of Databases and Information Systems, Ulm University, Germany

Permission is hereby granted, free of charge, to any person obtaining a copy 
of this software and associated documentation files (the "Software"), to deal 
in the Software without restriction, including without limitation the rights 
to use, copy, modify, merge, publish, distribute, sublicense, and/or sell 
copies of the Software, and to permit persons to whom the Software is 
furnished to do so, subject to the following conditions:

The above copyright notice and this permission notice shall be included in 
all copies or substantial portions of the Software.

THE SOFTWARE IS PROVIDED "AS IS", WITHOUT WARRANTY OF ANY KIND, EXPRESS OR 
IMPLIED, INCLUDING BUT NOT LIMITED TO THE WARRANTIES OF MERCHANTABILITY, 
FITNESS FOR A PARTICULAR PURPOSE AND NONINFRINGEMENT. IN NO EVENT SHALL THE 
AUTHORS OR COPYRIGHT HOLDERS BE LIABLE FOR ANY CLAIM, DAMAGES OR OTHER 
LIABILITY, WHETHER IN AN ACTION OF CONTRACT, TORT OR OTHERWISE, ARISING FROM, 
OUT OF OR IN CONNECTION WITH THE SOFTWARE OR THE USE OR OTHER DEALINGS 
IN THE SOFTWARE.
*)
IF NOT(fin) THEN
	IF TC.batchJobQueue.batchJobs[TC.currBatchJobIdx].workpieces[TC.batchJobQueue.batchJobs[TC.currBatchJobIdx].nextNotProcessedIdx].sortingLinePos = 1 THEN
		// go to eject point 1
		vg_move_to_pos(x := 25, y := 133, z := 2);
	ELSIF TC.batchJobQueue.batchJobs[TC.currBatchJobIdx].workpieces[TC.batchJobQueue.batchJobs[TC.currBatchJobIdx].nextNotProcessedIdx].sortingLinePos = 2 THEN
		// go to eject point 2
		vg_move_to_pos(x := 30, y := 133, z := 15);
	ELSE
		// go to eject point 3
		vg_move_to_pos(x := 49, y := 133, z := 23);
	END_IF
	fin := vg_move_to_pos.fin;
	IF fin THEN
		IF TC.batchJobQueue.batchJobs[TC.currBatchJobIdx].workpieces[TC.batchJobQueue.batchJobs[TC.currBatchJobIdx].nextNotProcessedIdx].sortingLinePos = 1 THEN
			VG.state := VG_State.AT_EJECT_1;
		ELSIF TC.batchJobQueue.batchJobs[TC.currBatchJobIdx].workpieces[TC.batchJobQueue.batchJobs[TC.currBatchJobIdx].nextNotProcessedIdx].sortingLinePos = 2 THEN
			VG.state := VG_State.AT_EJECT_2;
		ELSE
			VG.state := VG_State.AT_EJECT_3;
		END_IF
	END_IF
END_IF
END_ACTION

ACTION YDown_VG_DROP_W_active_exit:
(*
Copyright (c) 2019 Manuel Goester, Michael Witt, Klaus Kammerer
Institute of Databases and Information Systems, Ulm University, Germany

Permission is hereby granted, free of charge, to any person obtaining a copy 
of this software and associated documentation files (the "Software"), to deal 
in the Software without restriction, including without limitation the rights 
to use, copy, modify, merge, publish, distribute, sublicense, and/or sell 
copies of the Software, and to permit persons to whom the Software is 
furnished to do so, subject to the following conditions:

The above copyright notice and this permission notice shall be included in 
all copies or substantial portions of the Software.

THE SOFTWARE IS PROVIDED "AS IS", WITHOUT WARRANTY OF ANY KIND, EXPRESS OR 
IMPLIED, INCLUDING BUT NOT LIMITED TO THE WARRANTIES OF MERCHANTABILITY, 
FITNESS FOR A PARTICULAR PURPOSE AND NONINFRINGEMENT. IN NO EVENT SHALL THE 
AUTHORS OR COPYRIGHT HOLDERS BE LIABLE FOR ANY CLAIM, DAMAGES OR OTHER 
LIABILITY, WHETHER IN AN ACTION OF CONTRACT, TORT OR OTHERWISE, ARISING FROM, 
OUT OF OR IN CONNECTION WITH THE SOFTWARE OR THE USE OR OTHER DEALINGS 
IN THE SOFTWARE.
*)
yFin := FALSE;
END_ACTION

ACTION OpenVentil_VG_DROP_W_active_exit:
(*
Copyright (c) 2019 Manuel Goester, Michael Witt, Klaus Kammerer
Institute of Databases and Information Systems, Ulm University, Germany

Permission is hereby granted, free of charge, to any person obtaining a copy 
of this software and associated documentation files (the "Software"), to deal 
in the Software without restriction, including without limitation the rights 
to use, copy, modify, merge, publish, distribute, sublicense, and/or sell 
copies of the Software, and to permit persons to whom the Software is 
furnished to do so, subject to the following conditions:

The above copyright notice and this permission notice shall be included in 
all copies or substantial portions of the Software.

THE SOFTWARE IS PROVIDED "AS IS", WITHOUT WARRANTY OF ANY KIND, EXPRESS OR 
IMPLIED, INCLUDING BUT NOT LIMITED TO THE WARRANTIES OF MERCHANTABILITY, 
FITNESS FOR A PARTICULAR PURPOSE AND NONINFRINGEMENT. IN NO EVENT SHALL THE 
AUTHORS OR COPYRIGHT HOLDERS BE LIABLE FOR ANY CLAIM, DAMAGES OR OTHER 
LIABILITY, WHETHER IN AN ACTION OF CONTRACT, TORT OR OTHERWISE, ARISING FROM, 
OUT OF OR IN CONNECTION WITH THE SOFTWARE OR THE USE OR OTHER DEALINGS 
IN THE SOFTWARE.
*)
END_ACTION

ACTION VG_EJECT_W_active:
(*
Copyright (c) 2019 Manuel Goester, Michael Witt, Klaus Kammerer
Institute of Databases and Information Systems, Ulm University, Germany

Permission is hereby granted, free of charge, to any person obtaining a copy 
of this software and associated documentation files (the "Software"), to deal 
in the Software without restriction, including without limitation the rights 
to use, copy, modify, merge, publish, distribute, sublicense, and/or sell 
copies of the Software, and to permit persons to whom the Software is 
furnished to do so, subject to the following conditions:

The above copyright notice and this permission notice shall be included in 
all copies or substantial portions of the Software.

THE SOFTWARE IS PROVIDED "AS IS", WITHOUT WARRANTY OF ANY KIND, EXPRESS OR 
IMPLIED, INCLUDING BUT NOT LIMITED TO THE WARRANTIES OF MERCHANTABILITY, 
FITNESS FOR A PARTICULAR PURPOSE AND NONINFRINGEMENT. IN NO EVENT SHALL THE 
AUTHORS OR COPYRIGHT HOLDERS BE LIABLE FOR ANY CLAIM, DAMAGES OR OTHER 
LIABILITY, WHETHER IN AN ACTION OF CONTRACT, TORT OR OTHERWISE, ARISING FROM, 
OUT OF OR IN CONNECTION WITH THE SOFTWARE OR THE USE OR OTHER DEALINGS 
IN THE SOFTWARE.
*)
// Brings VG to its default pos where sVertical = sHorizontal = sRotation = 1
// 1. y-Axis 2. z-Axis 3. rotation
IF NOT(VG.sVertical) THEN
	VG.mVerticalUp := TRUE;
ELSE
	VG.mVerticalUp := FALSE;
	VG.cY := 0;
END_IF
IF NOT(VG.sHorizontal) THEN
	VG.mHorizontalBackward := TRUE;
ELSE
	VG.mHorizontalBackward := FALSE;
	VG.cX := 0;
END_IF
IF NOT(VG.sRotation) THEN
	VG.mRotationClockwise := TRUE;
ELSE
	VG.mRotationClockwise := FALSE;
	VG.cZ := 0;
END_IF

IF VG.sHorizontal AND VG.sVertical AND VG.sRotation THEN
	// default pos reached
	VG.state := VG_State.AT_DEFAULT_POS;
END_IF
END_ACTION

ACTION OpenVentil_VG_DROP_W_active_active:
(*
Copyright (c) 2019 Manuel Goester, Michael Witt, Klaus Kammerer
Institute of Databases and Information Systems, Ulm University, Germany

Permission is hereby granted, free of charge, to any person obtaining a copy 
of this software and associated documentation files (the "Software"), to deal 
in the Software without restriction, including without limitation the rights 
to use, copy, modify, merge, publish, distribute, sublicense, and/or sell 
copies of the Software, and to permit persons to whom the Software is 
furnished to do so, subject to the following conditions:

The above copyright notice and this permission notice shall be included in 
all copies or substantial portions of the Software.

THE SOFTWARE IS PROVIDED "AS IS", WITHOUT WARRANTY OF ANY KIND, EXPRESS OR 
IMPLIED, INCLUDING BUT NOT LIMITED TO THE WARRANTIES OF MERCHANTABILITY, 
FITNESS FOR A PARTICULAR PURPOSE AND NONINFRINGEMENT. IN NO EVENT SHALL THE 
AUTHORS OR COPYRIGHT HOLDERS BE LIABLE FOR ANY CLAIM, DAMAGES OR OTHER 
LIABILITY, WHETHER IN AN ACTION OF CONTRACT, TORT OR OTHERWISE, ARISING FROM, 
OUT OF OR IN CONNECTION WITH THE SOFTWARE OR THE USE OR OTHER DEALINGS 
IN THE SOFTWARE.
*)
VG.valve := FALSE;
pneumatic_loaded := FALSE;
END_ACTION

ACTION ZBack_VG_FROM_SL_TO_HR_active_active:
(*
Copyright (c) 2019 Manuel Goester, Michael Witt, Klaus Kammerer
Institute of Databases and Information Systems, Ulm University, Germany

Permission is hereby granted, free of charge, to any person obtaining a copy 
of this software and associated documentation files (the "Software"), to deal 
in the Software without restriction, including without limitation the rights 
to use, copy, modify, merge, publish, distribute, sublicense, and/or sell 
copies of the Software, and to permit persons to whom the Software is 
furnished to do so, subject to the following conditions:

The above copyright notice and this permission notice shall be included in 
all copies or substantial portions of the Software.

THE SOFTWARE IS PROVIDED "AS IS", WITHOUT WARRANTY OF ANY KIND, EXPRESS OR 
IMPLIED, INCLUDING BUT NOT LIMITED TO THE WARRANTIES OF MERCHANTABILITY, 
FITNESS FOR A PARTICULAR PURPOSE AND NONINFRINGEMENT. IN NO EVENT SHALL THE 
AUTHORS OR COPYRIGHT HOLDERS BE LIABLE FOR ANY CLAIM, DAMAGES OR OTHER 
LIABILITY, WHETHER IN AN ACTION OF CONTRACT, TORT OR OTHERWISE, ARISING FROM, 
OUT OF OR IN CONNECTION WITH THE SOFTWARE OR THE USE OR OTHER DEALINGS 
IN THE SOFTWARE.
*)
IF NOT(VG.sHorizontal) THEN
	VG.mHorizontalBackward := TRUE;
ELSE
	VG.mHorizontalBackward := FALSE;
	zFin := TRUE;
END_IF
END_ACTION

ACTION ZLeft_AND_XForward_VG_TO_FU_active_active:
(*
Copyright (c) 2019 Manuel Goester, Michael Witt, Klaus Kammerer
Institute of Databases and Information Systems, Ulm University, Germany

Permission is hereby granted, free of charge, to any person obtaining a copy 
of this software and associated documentation files (the "Software"), to deal 
in the Software without restriction, including without limitation the rights 
to use, copy, modify, merge, publish, distribute, sublicense, and/or sell 
copies of the Software, and to permit persons to whom the Software is 
furnished to do so, subject to the following conditions:

The above copyright notice and this permission notice shall be included in 
all copies or substantial portions of the Software.

THE SOFTWARE IS PROVIDED "AS IS", WITHOUT WARRANTY OF ANY KIND, EXPRESS OR 
IMPLIED, INCLUDING BUT NOT LIMITED TO THE WARRANTIES OF MERCHANTABILITY, 
FITNESS FOR A PARTICULAR PURPOSE AND NONINFRINGEMENT. IN NO EVENT SHALL THE 
AUTHORS OR COPYRIGHT HOLDERS BE LIABLE FOR ANY CLAIM, DAMAGES OR OTHER 
LIABILITY, WHETHER IN AN ACTION OF CONTRACT, TORT OR OTHERWISE, ARISING FROM, 
OUT OF OR IN CONNECTION WITH THE SOFTWARE OR THE USE OR OTHER DEALINGS 
IN THE SOFTWARE.
*)
IF NOT(fin) THEN
	vg_move_to_pos(x := 131, y := 0, z := 137);
	fin := vg_move_to_pos.fin;
END_IF
END_ACTION

ACTION YDown_VG_TAKE_W_active_exit:
(*
Copyright (c) 2019 Manuel Goester, Michael Witt, Klaus Kammerer
Institute of Databases and Information Systems, Ulm University, Germany

Permission is hereby granted, free of charge, to any person obtaining a copy 
of this software and associated documentation files (the "Software"), to deal 
in the Software without restriction, including without limitation the rights 
to use, copy, modify, merge, publish, distribute, sublicense, and/or sell 
copies of the Software, and to permit persons to whom the Software is 
furnished to do so, subject to the following conditions:

The above copyright notice and this permission notice shall be included in 
all copies or substantial portions of the Software.

THE SOFTWARE IS PROVIDED "AS IS", WITHOUT WARRANTY OF ANY KIND, EXPRESS OR 
IMPLIED, INCLUDING BUT NOT LIMITED TO THE WARRANTIES OF MERCHANTABILITY, 
FITNESS FOR A PARTICULAR PURPOSE AND NONINFRINGEMENT. IN NO EVENT SHALL THE 
AUTHORS OR COPYRIGHT HOLDERS BE LIABLE FOR ANY CLAIM, DAMAGES OR OTHER 
LIABILITY, WHETHER IN AN ACTION OF CONTRACT, TORT OR OTHERWISE, ARISING FROM, 
OUT OF OR IN CONNECTION WITH THE SOFTWARE OR THE USE OR OTHER DEALINGS 
IN THE SOFTWARE.
*)
yFin := FALSE;
END_ACTION

ACTION YUp_VG_TO_FU_active_exit:
(*
Copyright (c) 2019 Manuel Goester, Michael Witt, Klaus Kammerer
Institute of Databases and Information Systems, Ulm University, Germany

Permission is hereby granted, free of charge, to any person obtaining a copy 
of this software and associated documentation files (the "Software"), to deal 
in the Software without restriction, including without limitation the rights 
to use, copy, modify, merge, publish, distribute, sublicense, and/or sell 
copies of the Software, and to permit persons to whom the Software is 
furnished to do so, subject to the following conditions:

The above copyright notice and this permission notice shall be included in 
all copies or substantial portions of the Software.

THE SOFTWARE IS PROVIDED "AS IS", WITHOUT WARRANTY OF ANY KIND, EXPRESS OR 
IMPLIED, INCLUDING BUT NOT LIMITED TO THE WARRANTIES OF MERCHANTABILITY, 
FITNESS FOR A PARTICULAR PURPOSE AND NONINFRINGEMENT. IN NO EVENT SHALL THE 
AUTHORS OR COPYRIGHT HOLDERS BE LIABLE FOR ANY CLAIM, DAMAGES OR OTHER 
LIABILITY, WHETHER IN AN ACTION OF CONTRACT, TORT OR OTHERWISE, ARISING FROM, 
OUT OF OR IN CONNECTION WITH THE SOFTWARE OR THE USE OR OTHER DEALINGS 
IN THE SOFTWARE.
*)
yFin := FALSE;
VG.state := VG_State.TO_DEFAULT_POS;
SM.currW.state := W_State.AT_FUR_IN_WAGON;
VG_SINGLE_MODE.subBlockStart := FALSE;
END_ACTION

ACTION YUp_VG_TAKE_W_active_exit:
(*
Copyright (c) 2019 Manuel Goester, Michael Witt, Klaus Kammerer
Institute of Databases and Information Systems, Ulm University, Germany

Permission is hereby granted, free of charge, to any person obtaining a copy 
of this software and associated documentation files (the "Software"), to deal 
in the Software without restriction, including without limitation the rights 
to use, copy, modify, merge, publish, distribute, sublicense, and/or sell 
copies of the Software, and to permit persons to whom the Software is 
furnished to do so, subject to the following conditions:

The above copyright notice and this permission notice shall be included in 
all copies or substantial portions of the Software.

THE SOFTWARE IS PROVIDED "AS IS", WITHOUT WARRANTY OF ANY KIND, EXPRESS OR 
IMPLIED, INCLUDING BUT NOT LIMITED TO THE WARRANTIES OF MERCHANTABILITY, 
FITNESS FOR A PARTICULAR PURPOSE AND NONINFRINGEMENT. IN NO EVENT SHALL THE 
AUTHORS OR COPYRIGHT HOLDERS BE LIABLE FOR ANY CLAIM, DAMAGES OR OTHER 
LIABILITY, WHETHER IN AN ACTION OF CONTRACT, TORT OR OTHERWISE, ARISING FROM, 
OUT OF OR IN CONNECTION WITH THE SOFTWARE OR THE USE OR OTHER DEALINGS 
IN THE SOFTWARE.
*)
// reset flag
yFin := FALSE;
// workpiece is now at VG
SM.currW.linePos := 1;
// reset flag
VG_SINGLE_MODE.subBlockStart := FALSE;

// set HR state
HR.state := HR_State.AT_CONVEYOR_BOX_EMPTY;

IF SM.currW.format.ejectEnabled AND NOT(SM.currW.format.furEnabled) AND NOT(SM.currW.format.sawEnabled) AND NOT(SM.currW.format.colorCheckEnabled) THEN
	// directly eject workpiece
	VG.state := VG_State.FROM_HR_TO_EJECT;
ELSE
	// bring workpiece to FUR
	VG.state := VG_State.FROM_HR_TO_FUR;
END_IF
END_ACTION

ACTION Init_active:
(*
Copyright (c) 2019 Manuel Goester, Michael Witt, Klaus Kammerer
Institute of Databases and Information Systems, Ulm University, Germany

Permission is hereby granted, free of charge, to any person obtaining a copy 
of this software and associated documentation files (the "Software"), to deal 
in the Software without restriction, including without limitation the rights 
to use, copy, modify, merge, publish, distribute, sublicense, and/or sell 
copies of the Software, and to permit persons to whom the Software is 
furnished to do so, subject to the following conditions:

The above copyright notice and this permission notice shall be included in 
all copies or substantial portions of the Software.

THE SOFTWARE IS PROVIDED "AS IS", WITHOUT WARRANTY OF ANY KIND, EXPRESS OR 
IMPLIED, INCLUDING BUT NOT LIMITED TO THE WARRANTIES OF MERCHANTABILITY, 
FITNESS FOR A PARTICULAR PURPOSE AND NONINFRINGEMENT. IN NO EVENT SHALL THE 
AUTHORS OR COPYRIGHT HOLDERS BE LIABLE FOR ANY CLAIM, DAMAGES OR OTHER 
LIABILITY, WHETHER IN AN ACTION OF CONTRACT, TORT OR OTHERWISE, ARISING FROM, 
OUT OF OR IN CONNECTION WITH THE SOFTWARE OR THE USE OR OTHER DEALINGS 
IN THE SOFTWARE.
*)
subBlockStart := FALSE;
END_ACTION

ACTION YDown_VG_TO_FU_active_active:
(*
Copyright (c) 2019 Manuel Goester, Michael Witt, Klaus Kammerer
Institute of Databases and Information Systems, Ulm University, Germany

Permission is hereby granted, free of charge, to any person obtaining a copy 
of this software and associated documentation files (the "Software"), to deal 
in the Software without restriction, including without limitation the rights 
to use, copy, modify, merge, publish, distribute, sublicense, and/or sell 
copies of the Software, and to permit persons to whom the Software is 
furnished to do so, subject to the following conditions:

The above copyright notice and this permission notice shall be included in 
all copies or substantial portions of the Software.

THE SOFTWARE IS PROVIDED "AS IS", WITHOUT WARRANTY OF ANY KIND, EXPRESS OR 
IMPLIED, INCLUDING BUT NOT LIMITED TO THE WARRANTIES OF MERCHANTABILITY, 
FITNESS FOR A PARTICULAR PURPOSE AND NONINFRINGEMENT. IN NO EVENT SHALL THE 
AUTHORS OR COPYRIGHT HOLDERS BE LIABLE FOR ANY CLAIM, DAMAGES OR OTHER 
LIABILITY, WHETHER IN AN ACTION OF CONTRACT, TORT OR OTHERWISE, ARISING FROM, 
OUT OF OR IN CONNECTION WITH THE SOFTWARE OR THE USE OR OTHER DEALINGS 
IN THE SOFTWARE.
*)
IF NOT(fin) THEN
	vg_move_to_pos(x := 131, y := 85, z := 137);
	fin := vg_move_to_pos.fin;
END_IF
END_ACTION

ACTION ZBack_VG_TO_FU_active_exit:
(*
Copyright (c) 2019 Manuel Goester, Michael Witt, Klaus Kammerer
Institute of Databases and Information Systems, Ulm University, Germany

Permission is hereby granted, free of charge, to any person obtaining a copy 
of this software and associated documentation files (the "Software"), to deal 
in the Software without restriction, including without limitation the rights 
to use, copy, modify, merge, publish, distribute, sublicense, and/or sell 
copies of the Software, and to permit persons to whom the Software is 
furnished to do so, subject to the following conditions:

The above copyright notice and this permission notice shall be included in 
all copies or substantial portions of the Software.

THE SOFTWARE IS PROVIDED "AS IS", WITHOUT WARRANTY OF ANY KIND, EXPRESS OR 
IMPLIED, INCLUDING BUT NOT LIMITED TO THE WARRANTIES OF MERCHANTABILITY, 
FITNESS FOR A PARTICULAR PURPOSE AND NONINFRINGEMENT. IN NO EVENT SHALL THE 
AUTHORS OR COPYRIGHT HOLDERS BE LIABLE FOR ANY CLAIM, DAMAGES OR OTHER 
LIABILITY, WHETHER IN AN ACTION OF CONTRACT, TORT OR OTHERWISE, ARISING FROM, 
OUT OF OR IN CONNECTION WITH THE SOFTWARE OR THE USE OR OTHER DEALINGS 
IN THE SOFTWARE.
*)
zFin := FALSE;
END_ACTION

ACTION YUp_VG_TO_FU_active_active:
(*
Copyright (c) 2019 Manuel Goester, Michael Witt, Klaus Kammerer
Institute of Databases and Information Systems, Ulm University, Germany

Permission is hereby granted, free of charge, to any person obtaining a copy 
of this software and associated documentation files (the "Software"), to deal 
in the Software without restriction, including without limitation the rights 
to use, copy, modify, merge, publish, distribute, sublicense, and/or sell 
copies of the Software, and to permit persons to whom the Software is 
furnished to do so, subject to the following conditions:

The above copyright notice and this permission notice shall be included in 
all copies or substantial portions of the Software.

THE SOFTWARE IS PROVIDED "AS IS", WITHOUT WARRANTY OF ANY KIND, EXPRESS OR 
IMPLIED, INCLUDING BUT NOT LIMITED TO THE WARRANTIES OF MERCHANTABILITY, 
FITNESS FOR A PARTICULAR PURPOSE AND NONINFRINGEMENT. IN NO EVENT SHALL THE 
AUTHORS OR COPYRIGHT HOLDERS BE LIABLE FOR ANY CLAIM, DAMAGES OR OTHER 
LIABILITY, WHETHER IN AN ACTION OF CONTRACT, TORT OR OTHERWISE, ARISING FROM, 
OUT OF OR IN CONNECTION WITH THE SOFTWARE OR THE USE OR OTHER DEALINGS 
IN THE SOFTWARE.
*)
IF NOT(VG.sVertical) THEN
	VG.mVerticalUp := TRUE;
ELSE
	VG.mVerticalUp := FALSE;
	VG.cY := 0;
	yFin := TRUE;
END_IF
END_ACTION

ACTION ZBack_VG_TAKE_W_active_exit:
(*
Copyright (c) 2019 Manuel Goester, Michael Witt, Klaus Kammerer
Institute of Databases and Information Systems, Ulm University, Germany

Permission is hereby granted, free of charge, to any person obtaining a copy 
of this software and associated documentation files (the "Software"), to deal 
in the Software without restriction, including without limitation the rights 
to use, copy, modify, merge, publish, distribute, sublicense, and/or sell 
copies of the Software, and to permit persons to whom the Software is 
furnished to do so, subject to the following conditions:

The above copyright notice and this permission notice shall be included in 
all copies or substantial portions of the Software.

THE SOFTWARE IS PROVIDED "AS IS", WITHOUT WARRANTY OF ANY KIND, EXPRESS OR 
IMPLIED, INCLUDING BUT NOT LIMITED TO THE WARRANTIES OF MERCHANTABILITY, 
FITNESS FOR A PARTICULAR PURPOSE AND NONINFRINGEMENT. IN NO EVENT SHALL THE 
AUTHORS OR COPYRIGHT HOLDERS BE LIABLE FOR ANY CLAIM, DAMAGES OR OTHER 
LIABILITY, WHETHER IN AN ACTION OF CONTRACT, TORT OR OTHERWISE, ARISING FROM, 
OUT OF OR IN CONNECTION WITH THE SOFTWARE OR THE USE OR OTHER DEALINGS 
IN THE SOFTWARE.
*)
zFin := FALSE;
END_ACTION

ACTION VG_TO_FU_active:
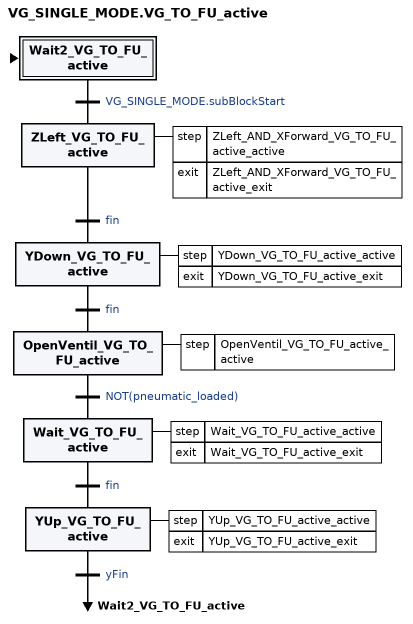
INITIAL_STEP Wait2_VG_TO_FU_active:
END_STEP
TRANSITION FROM Wait2_VG_TO_FU_active TO ZLeft_VG_TO_FU_active
    := VG_SINGLE_MODE.subBlockStart;
END_TRANSITION
STEP ZLeft_VG_TO_FU_active:
    ZLeft_AND_XForward_VG_TO_FU_active_active(N);  // step action
    ZLeft_AND_XForward_VG_TO_FU_active_exit(P0);  // exit action
END_STEP
TRANSITION FROM ZLeft_VG_TO_FU_active TO YDown_VG_TO_FU_active
    := fin;
END_TRANSITION
STEP YDown_VG_TO_FU_active:
    YDown_VG_TO_FU_active_active(N);  // step action
    YDown_VG_TO_FU_active_exit(P0);  // exit action
END_STEP
TRANSITION FROM YDown_VG_TO_FU_active TO OpenVentil_VG_TO_FU_active
    := fin;
END_TRANSITION
STEP OpenVentil_VG_TO_FU_active:
    OpenVentil_VG_TO_FU_active_active(N);  // step action
END_STEP
TRANSITION FROM OpenVentil_VG_TO_FU_active TO Wait_VG_TO_FU_active
    := NOT(pneumatic_loaded);
END_TRANSITION
STEP Wait_VG_TO_FU_active:
    Wait_VG_TO_FU_active_active(N);  // step action
    Wait_VG_TO_FU_active_exit(P0);  // exit action
END_STEP
TRANSITION FROM Wait_VG_TO_FU_active TO YUp_VG_TO_FU_active
    := fin;
END_TRANSITION
STEP YUp_VG_TO_FU_active:
    YUp_VG_TO_FU_active_active(N);  // step action
    YUp_VG_TO_FU_active_exit(P0);  // exit action
END_STEP
TRANSITION FROM YUp_VG_TO_FU_active TO Wait2_VG_TO_FU_active
    := yFin;
END_TRANSITION
END_ACTION

ACTION OpenVentil_VG_TO_FU_active_active:
(*
Copyright (c) 2019 Manuel Goester, Michael Witt, Klaus Kammerer
Institute of Databases and Information Systems, Ulm University, Germany

Permission is hereby granted, free of charge, to any person obtaining a copy 
of this software and associated documentation files (the "Software"), to deal 
in the Software without restriction, including without limitation the rights 
to use, copy, modify, merge, publish, distribute, sublicense, and/or sell 
copies of the Software, and to permit persons to whom the Software is 
furnished to do so, subject to the following conditions:

The above copyright notice and this permission notice shall be included in 
all copies or substantial portions of the Software.

THE SOFTWARE IS PROVIDED "AS IS", WITHOUT WARRANTY OF ANY KIND, EXPRESS OR 
IMPLIED, INCLUDING BUT NOT LIMITED TO THE WARRANTIES OF MERCHANTABILITY, 
FITNESS FOR A PARTICULAR PURPOSE AND NONINFRINGEMENT. IN NO EVENT SHALL THE 
AUTHORS OR COPYRIGHT HOLDERS BE LIABLE FOR ANY CLAIM, DAMAGES OR OTHER 
LIABILITY, WHETHER IN AN ACTION OF CONTRACT, TORT OR OTHERWISE, ARISING FROM, 
OUT OF OR IN CONNECTION WITH THE SOFTWARE OR THE USE OR OTHER DEALINGS 
IN THE SOFTWARE.
*)
VG.valve := FALSE;
pneumatic_loaded := FALSE;
END_ACTION

ACTION YUp_VG_DROP_W_active_active:
(*
Copyright (c) 2019 Manuel Goester, Michael Witt, Klaus Kammerer
Institute of Databases and Information Systems, Ulm University, Germany

Permission is hereby granted, free of charge, to any person obtaining a copy 
of this software and associated documentation files (the "Software"), to deal 
in the Software without restriction, including without limitation the rights 
to use, copy, modify, merge, publish, distribute, sublicense, and/or sell 
copies of the Software, and to permit persons to whom the Software is 
furnished to do so, subject to the following conditions:

The above copyright notice and this permission notice shall be included in 
all copies or substantial portions of the Software.

THE SOFTWARE IS PROVIDED "AS IS", WITHOUT WARRANTY OF ANY KIND, EXPRESS OR 
IMPLIED, INCLUDING BUT NOT LIMITED TO THE WARRANTIES OF MERCHANTABILITY, 
FITNESS FOR A PARTICULAR PURPOSE AND NONINFRINGEMENT. IN NO EVENT SHALL THE 
AUTHORS OR COPYRIGHT HOLDERS BE LIABLE FOR ANY CLAIM, DAMAGES OR OTHER 
LIABILITY, WHETHER IN AN ACTION OF CONTRACT, TORT OR OTHERWISE, ARISING FROM, 
OUT OF OR IN CONNECTION WITH THE SOFTWARE OR THE USE OR OTHER DEALINGS 
IN THE SOFTWARE.
*)
HR.state := HR_State.AT_CONVEYOR_BOX_FULL;
IF NOT(VG.sVertical) THEN
	VG.mVerticalUp := TRUE;
ELSE
	VG.mVerticalUp := FALSE;
	VG.cY := 0;
	yFin := TRUE;
END_IF
END_ACTION

ACTION ZBack_VG_TAKE_W_active_active:
(*
Copyright (c) 2019 Manuel Goester, Michael Witt, Klaus Kammerer
Institute of Databases and Information Systems, Ulm University, Germany

Permission is hereby granted, free of charge, to any person obtaining a copy 
of this software and associated documentation files (the "Software"), to deal 
in the Software without restriction, including without limitation the rights 
to use, copy, modify, merge, publish, distribute, sublicense, and/or sell 
copies of the Software, and to permit persons to whom the Software is 
furnished to do so, subject to the following conditions:

The above copyright notice and this permission notice shall be included in 
all copies or substantial portions of the Software.

THE SOFTWARE IS PROVIDED "AS IS", WITHOUT WARRANTY OF ANY KIND, EXPRESS OR 
IMPLIED, INCLUDING BUT NOT LIMITED TO THE WARRANTIES OF MERCHANTABILITY, 
FITNESS FOR A PARTICULAR PURPOSE AND NONINFRINGEMENT. IN NO EVENT SHALL THE 
AUTHORS OR COPYRIGHT HOLDERS BE LIABLE FOR ANY CLAIM, DAMAGES OR OTHER 
LIABILITY, WHETHER IN AN ACTION OF CONTRACT, TORT OR OTHERWISE, ARISING FROM, 
OUT OF OR IN CONNECTION WITH THE SOFTWARE OR THE USE OR OTHER DEALINGS 
IN THE SOFTWARE.
*)
IF NOT(VG.sHorizontal) THEN
	VG.mHorizontalBackward := TRUE;
ELSE
	VG.mHorizontalBackward := FALSE;
	
END_IF
END_ACTION

ACTION VG_TAKE_W_entry:
(*
Copyright (c) 2019 Manuel Goester, Michael Witt, Klaus Kammerer
Institute of Databases and Information Systems, Ulm University, Germany

Permission is hereby granted, free of charge, to any person obtaining a copy 
of this software and associated documentation files (the "Software"), to deal 
in the Software without restriction, including without limitation the rights 
to use, copy, modify, merge, publish, distribute, sublicense, and/or sell 
copies of the Software, and to permit persons to whom the Software is 
furnished to do so, subject to the following conditions:

The above copyright notice and this permission notice shall be included in 
all copies or substantial portions of the Software.

THE SOFTWARE IS PROVIDED "AS IS", WITHOUT WARRANTY OF ANY KIND, EXPRESS OR 
IMPLIED, INCLUDING BUT NOT LIMITED TO THE WARRANTIES OF MERCHANTABILITY, 
FITNESS FOR A PARTICULAR PURPOSE AND NONINFRINGEMENT. IN NO EVENT SHALL THE 
AUTHORS OR COPYRIGHT HOLDERS BE LIABLE FOR ANY CLAIM, DAMAGES OR OTHER 
LIABILITY, WHETHER IN AN ACTION OF CONTRACT, TORT OR OTHERWISE, ARISING FROM, 
OUT OF OR IN CONNECTION WITH THE SOFTWARE OR THE USE OR OTHER DEALINGS 
IN THE SOFTWARE.
*)
VG_SINGLE_MODE.subBlockStart := TRUE;
END_ACTION

ACTION Wait_VG_TO_FU_active_active:
(*
Copyright (c) 2019 Manuel Goester, Michael Witt, Klaus Kammerer
Institute of Databases and Information Systems, Ulm University, Germany

Permission is hereby granted, free of charge, to any person obtaining a copy 
of this software and associated documentation files (the "Software"), to deal 
in the Software without restriction, including without limitation the rights 
to use, copy, modify, merge, publish, distribute, sublicense, and/or sell 
copies of the Software, and to permit persons to whom the Software is 
furnished to do so, subject to the following conditions:

The above copyright notice and this permission notice shall be included in 
all copies or substantial portions of the Software.

THE SOFTWARE IS PROVIDED "AS IS", WITHOUT WARRANTY OF ANY KIND, EXPRESS OR 
IMPLIED, INCLUDING BUT NOT LIMITED TO THE WARRANTIES OF MERCHANTABILITY, 
FITNESS FOR A PARTICULAR PURPOSE AND NONINFRINGEMENT. IN NO EVENT SHALL THE 
AUTHORS OR COPYRIGHT HOLDERS BE LIABLE FOR ANY CLAIM, DAMAGES OR OTHER 
LIABILITY, WHETHER IN AN ACTION OF CONTRACT, TORT OR OTHERWISE, ARISING FROM, 
OUT OF OR IN CONNECTION WITH THE SOFTWARE OR THE USE OR OTHER DEALINGS 
IN THE SOFTWARE.
*)
timer(IN:= TRUE, PT:= T#1S);
IF NOT(timer.Q = FALSE AND timer.IN) THEN
	// reset timer
	timer(IN:= FALSE);
	// go to next step
	fin := TRUE;
END_IF
END_ACTION

ACTION YUp_VG_TAKE_W_active_active:
(*
Copyright (c) 2019 Manuel Goester, Michael Witt, Klaus Kammerer
Institute of Databases and Information Systems, Ulm University, Germany

Permission is hereby granted, free of charge, to any person obtaining a copy 
of this software and associated documentation files (the "Software"), to deal 
in the Software without restriction, including without limitation the rights 
to use, copy, modify, merge, publish, distribute, sublicense, and/or sell 
copies of the Software, and to permit persons to whom the Software is 
furnished to do so, subject to the following conditions:

The above copyright notice and this permission notice shall be included in 
all copies or substantial portions of the Software.

THE SOFTWARE IS PROVIDED "AS IS", WITHOUT WARRANTY OF ANY KIND, EXPRESS OR 
IMPLIED, INCLUDING BUT NOT LIMITED TO THE WARRANTIES OF MERCHANTABILITY, 
FITNESS FOR A PARTICULAR PURPOSE AND NONINFRINGEMENT. IN NO EVENT SHALL THE 
AUTHORS OR COPYRIGHT HOLDERS BE LIABLE FOR ANY CLAIM, DAMAGES OR OTHER 
LIABILITY, WHETHER IN AN ACTION OF CONTRACT, TORT OR OTHERWISE, ARISING FROM, 
OUT OF OR IN CONNECTION WITH THE SOFTWARE OR THE USE OR OTHER DEALINGS 
IN THE SOFTWARE.
*)
IF NOT(VG.sVertical) THEN
	VG.mVerticalUp := TRUE;
ELSE
	VG.mVerticalUp := FALSE;
	VG.cY := 0;
	yFin := TRUE;
END_IF
END_ACTION

ACTION VG_DROP_W_entry:
(*
Copyright (c) 2019 Manuel Goester, Michael Witt, Klaus Kammerer
Institute of Databases and Information Systems, Ulm University, Germany

Permission is hereby granted, free of charge, to any person obtaining a copy 
of this software and associated documentation files (the "Software"), to deal 
in the Software without restriction, including without limitation the rights 
to use, copy, modify, merge, publish, distribute, sublicense, and/or sell 
copies of the Software, and to permit persons to whom the Software is 
furnished to do so, subject to the following conditions:

The above copyright notice and this permission notice shall be included in 
all copies or substantial portions of the Software.

THE SOFTWARE IS PROVIDED "AS IS", WITHOUT WARRANTY OF ANY KIND, EXPRESS OR 
IMPLIED, INCLUDING BUT NOT LIMITED TO THE WARRANTIES OF MERCHANTABILITY, 
FITNESS FOR A PARTICULAR PURPOSE AND NONINFRINGEMENT. IN NO EVENT SHALL THE 
AUTHORS OR COPYRIGHT HOLDERS BE LIABLE FOR ANY CLAIM, DAMAGES OR OTHER 
LIABILITY, WHETHER IN AN ACTION OF CONTRACT, TORT OR OTHERWISE, ARISING FROM, 
OUT OF OR IN CONNECTION WITH THE SOFTWARE OR THE USE OR OTHER DEALINGS 
IN THE SOFTWARE.
*)
VG_SINGLE_MODE.subBlockStart := TRUE;
END_ACTION

ACTION VG_TO_DEFAULT_POS_active:
(*
Copyright (c) 2019 Manuel Goester, Michael Witt, Klaus Kammerer
Institute of Databases and Information Systems, Ulm University, Germany

Permission is hereby granted, free of charge, to any person obtaining a copy 
of this software and associated documentation files (the "Software"), to deal 
in the Software without restriction, including without limitation the rights 
to use, copy, modify, merge, publish, distribute, sublicense, and/or sell 
copies of the Software, and to permit persons to whom the Software is 
furnished to do so, subject to the following conditions:

The above copyright notice and this permission notice shall be included in 
all copies or substantial portions of the Software.

THE SOFTWARE IS PROVIDED "AS IS", WITHOUT WARRANTY OF ANY KIND, EXPRESS OR 
IMPLIED, INCLUDING BUT NOT LIMITED TO THE WARRANTIES OF MERCHANTABILITY, 
FITNESS FOR A PARTICULAR PURPOSE AND NONINFRINGEMENT. IN NO EVENT SHALL THE 
AUTHORS OR COPYRIGHT HOLDERS BE LIABLE FOR ANY CLAIM, DAMAGES OR OTHER 
LIABILITY, WHETHER IN AN ACTION OF CONTRACT, TORT OR OTHERWISE, ARISING FROM, 
OUT OF OR IN CONNECTION WITH THE SOFTWARE OR THE USE OR OTHER DEALINGS 
IN THE SOFTWARE.
*)
// Brings VG to its default pos where sVertical = sHorizontal = sRotation = 1
// 1. y-Axis 2. z-Axis 3. rotation
(*IF NOT(VG.sVertical) THEN
	VG.mVerticalUp := TRUE;
ELSE
	VG.mVerticalUp := FALSE;
	IF NOT(VG.sHorizontal) THEN
		VG.mHorizontalBackward := TRUE;
	ELSE
		VG.mHorizontalBackward := FALSE;
		IF NOT(VG.sRotation) THEN
			VG.mRotationClockwise := TRUE;
		ELSE
			VG.mRotationClockwise := FALSE;
			// default pos reached
			VG.state := VG_State.AT_DEFAULT_POS;
			VG.cX := 0;
			VG.cY := 0;
			VG.cZ := 0;
		END_IF
	END_IF
END_IF *)
VG.state := VG_State.AT_DEFAULT_POS;
END_ACTION

ACTION VG_DROP_W_active:
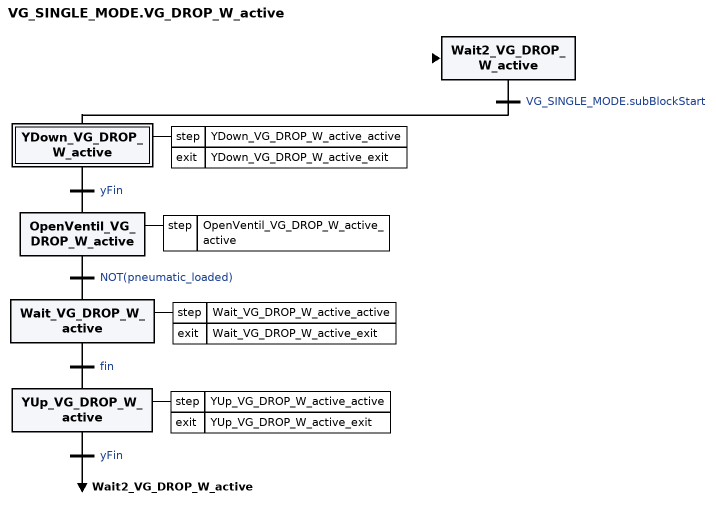
STEP Wait2_VG_DROP_W_active:
END_STEP
TRANSITION FROM Wait2_VG_DROP_W_active TO YDown_VG_DROP_W_active
    := VG_SINGLE_MODE.subBlockStart;
END_TRANSITION
INITIAL_STEP YDown_VG_DROP_W_active:
    YDown_VG_DROP_W_active_active(N);  // step action
    YDown_VG_DROP_W_active_exit(P0);  // exit action
END_STEP
TRANSITION FROM YDown_VG_DROP_W_active TO OpenVentil_VG_DROP_W_active
    := yFin;
END_TRANSITION
STEP OpenVentil_VG_DROP_W_active:
    OpenVentil_VG_DROP_W_active_active(N);  // step action
END_STEP
TRANSITION FROM OpenVentil_VG_DROP_W_active TO Wait_VG_DROP_W_active
    := NOT(pneumatic_loaded);
END_TRANSITION
STEP Wait_VG_DROP_W_active:
    Wait_VG_DROP_W_active_active(N);  // step action
    Wait_VG_DROP_W_active_exit(P0);  // exit action
END_STEP
TRANSITION FROM Wait_VG_DROP_W_active TO YUp_VG_DROP_W_active
    := fin;
END_TRANSITION
STEP YUp_VG_DROP_W_active:
    YUp_VG_DROP_W_active_active(N);  // step action
    YUp_VG_DROP_W_active_exit(P0);  // exit action
END_STEP
TRANSITION FROM YUp_VG_DROP_W_active TO Wait2_VG_DROP_W_active
    := yFin;
END_TRANSITION
END_ACTION

ACTION VG_TAKE_W_active:
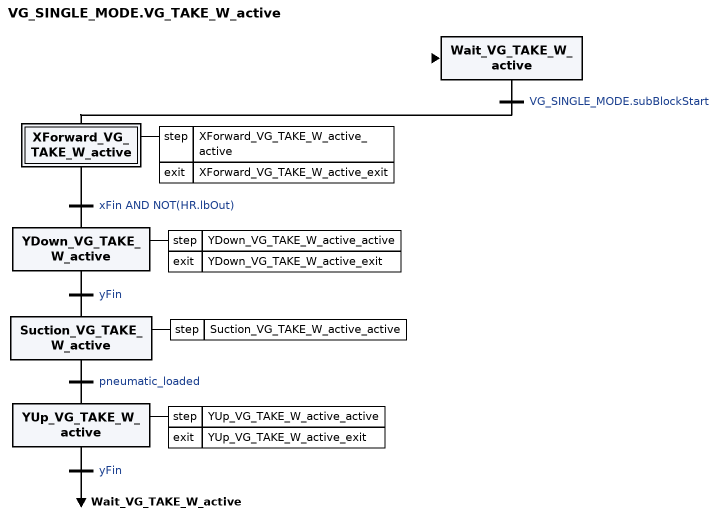
STEP Wait_VG_TAKE_W_active:
END_STEP
TRANSITION FROM Wait_VG_TAKE_W_active TO XForward_VG_TAKE_W_active
    := VG_SINGLE_MODE.subBlockStart;
END_TRANSITION
INITIAL_STEP XForward_VG_TAKE_W_active:
    XForward_VG_TAKE_W_active_active(N);  // step action
    XForward_VG_TAKE_W_active_exit(P0);  // exit action
END_STEP
TRANSITION FROM XForward_VG_TAKE_W_active TO YDown_VG_TAKE_W_active
    := xFin AND NOT(HR.lbOut);
END_TRANSITION
STEP YDown_VG_TAKE_W_active:
    YDown_VG_TAKE_W_active_active(N);  // step action
    YDown_VG_TAKE_W_active_exit(P0);  // exit action
END_STEP
TRANSITION FROM YDown_VG_TAKE_W_active TO Suction_VG_TAKE_W_active
    := yFin;
END_TRANSITION
STEP Suction_VG_TAKE_W_active:
    Suction_VG_TAKE_W_active_active(N);  // step action
END_STEP
TRANSITION FROM Suction_VG_TAKE_W_active TO YUp_VG_TAKE_W_active
    := pneumatic_loaded;
END_TRANSITION
STEP YUp_VG_TAKE_W_active:
    YUp_VG_TAKE_W_active_active(N);  // step action
    YUp_VG_TAKE_W_active_exit(P0);  // exit action
END_STEP
TRANSITION FROM YUp_VG_TAKE_W_active TO Wait_VG_TAKE_W_active
    := yFin;
END_TRANSITION
END_ACTION

ACTION YDown_VG_TAKE_W_active_active:
(*
Copyright (c) 2019 Manuel Goester, Michael Witt, Klaus Kammerer
Institute of Databases and Information Systems, Ulm University, Germany

Permission is hereby granted, free of charge, to any person obtaining a copy 
of this software and associated documentation files (the "Software"), to deal 
in the Software without restriction, including without limitation the rights 
to use, copy, modify, merge, publish, distribute, sublicense, and/or sell 
copies of the Software, and to permit persons to whom the Software is 
furnished to do so, subject to the following conditions:

The above copyright notice and this permission notice shall be included in 
all copies or substantial portions of the Software.

THE SOFTWARE IS PROVIDED "AS IS", WITHOUT WARRANTY OF ANY KIND, EXPRESS OR 
IMPLIED, INCLUDING BUT NOT LIMITED TO THE WARRANTIES OF MERCHANTABILITY, 
FITNESS FOR A PARTICULAR PURPOSE AND NONINFRINGEMENT. IN NO EVENT SHALL THE 
AUTHORS OR COPYRIGHT HOLDERS BE LIABLE FOR ANY CLAIM, DAMAGES OR OTHER 
LIABILITY, WHETHER IN AN ACTION OF CONTRACT, TORT OR OTHERWISE, ARISING FROM, 
OUT OF OR IN CONNECTION WITH THE SOFTWARE OR THE USE OR OTHER DEALINGS 
IN THE SOFTWARE.
*)
IF NOT(yFin) THEN
	vg_move_to_pos(x:=27, y:=40, z:=206);
	yFin := vg_move_to_pos.fin;
END_IF
END_ACTION

ACTION Wait_VG_DROP_W_active_exit:
(*
Copyright (c) 2019 Manuel Goester, Michael Witt, Klaus Kammerer
Institute of Databases and Information Systems, Ulm University, Germany

Permission is hereby granted, free of charge, to any person obtaining a copy 
of this software and associated documentation files (the "Software"), to deal 
in the Software without restriction, including without limitation the rights 
to use, copy, modify, merge, publish, distribute, sublicense, and/or sell 
copies of the Software, and to permit persons to whom the Software is 
furnished to do so, subject to the following conditions:

The above copyright notice and this permission notice shall be included in 
all copies or substantial portions of the Software.

THE SOFTWARE IS PROVIDED "AS IS", WITHOUT WARRANTY OF ANY KIND, EXPRESS OR 
IMPLIED, INCLUDING BUT NOT LIMITED TO THE WARRANTIES OF MERCHANTABILITY, 
FITNESS FOR A PARTICULAR PURPOSE AND NONINFRINGEMENT. IN NO EVENT SHALL THE 
AUTHORS OR COPYRIGHT HOLDERS BE LIABLE FOR ANY CLAIM, DAMAGES OR OTHER 
LIABILITY, WHETHER IN AN ACTION OF CONTRACT, TORT OR OTHERWISE, ARISING FROM, 
OUT OF OR IN CONNECTION WITH THE SOFTWARE OR THE USE OR OTHER DEALINGS 
IN THE SOFTWARE.
*)
fin := FALSE;
END_ACTION

ACTION VG_DROP_W_exit:
(*
Copyright (c) 2019 Manuel Goester, Michael Witt, Klaus Kammerer
Institute of Databases and Information Systems, Ulm University, Germany

Permission is hereby granted, free of charge, to any person obtaining a copy 
of this software and associated documentation files (the "Software"), to deal 
in the Software without restriction, including without limitation the rights 
to use, copy, modify, merge, publish, distribute, sublicense, and/or sell 
copies of the Software, and to permit persons to whom the Software is 
furnished to do so, subject to the following conditions:

The above copyright notice and this permission notice shall be included in 
all copies or substantial portions of the Software.

THE SOFTWARE IS PROVIDED "AS IS", WITHOUT WARRANTY OF ANY KIND, EXPRESS OR 
IMPLIED, INCLUDING BUT NOT LIMITED TO THE WARRANTIES OF MERCHANTABILITY, 
FITNESS FOR A PARTICULAR PURPOSE AND NONINFRINGEMENT. IN NO EVENT SHALL THE 
AUTHORS OR COPYRIGHT HOLDERS BE LIABLE FOR ANY CLAIM, DAMAGES OR OTHER 
LIABILITY, WHETHER IN AN ACTION OF CONTRACT, TORT OR OTHERWISE, ARISING FROM, 
OUT OF OR IN CONNECTION WITH THE SOFTWARE OR THE USE OR OTHER DEALINGS 
IN THE SOFTWARE.
*)
VG_SINGLE_MODE.subBlockStart := FALSE;
END_ACTION

ACTION VG_FROM_SL_TO_HR_active:
(*
Copyright (c) 2019 Manuel Goester, Michael Witt, Klaus Kammerer
Institute of Databases and Information Systems, Ulm University, Germany

Permission is hereby granted, free of charge, to any person obtaining a copy 
of this software and associated documentation files (the "Software"), to deal 
in the Software without restriction, including without limitation the rights 
to use, copy, modify, merge, publish, distribute, sublicense, and/or sell 
copies of the Software, and to permit persons to whom the Software is 
furnished to do so, subject to the following conditions:

The above copyright notice and this permission notice shall be included in 
all copies or substantial portions of the Software.

THE SOFTWARE IS PROVIDED "AS IS", WITHOUT WARRANTY OF ANY KIND, EXPRESS OR 
IMPLIED, INCLUDING BUT NOT LIMITED TO THE WARRANTIES OF MERCHANTABILITY, 
FITNESS FOR A PARTICULAR PURPOSE AND NONINFRINGEMENT. IN NO EVENT SHALL THE 
AUTHORS OR COPYRIGHT HOLDERS BE LIABLE FOR ANY CLAIM, DAMAGES OR OTHER 
LIABILITY, WHETHER IN AN ACTION OF CONTRACT, TORT OR OTHERWISE, ARISING FROM, 
OUT OF OR IN CONNECTION WITH THE SOFTWARE OR THE USE OR OTHER DEALINGS 
IN THE SOFTWARE.
*)
// as long as VG is not at HR, it is going to HR
IF NOT(VG.state = VG_State.AT_HR) THEN
	VG.state := VG_State.FROM_SL_TO_HR;
	vg_move_to_pos(x := 27, y := 0, z := 206);
	IF vg_move_to_pos.fin THEN
		VG.state := VG_State.AT_HR;
	END_IF
END_IF
END_ACTION

ACTION VG_TO_HR_active:
(*
Copyright (c) 2019 Manuel Goester, Michael Witt, Klaus Kammerer
Institute of Databases and Information Systems, Ulm University, Germany

Permission is hereby granted, free of charge, to any person obtaining a copy 
of this software and associated documentation files (the "Software"), to deal 
in the Software without restriction, including without limitation the rights 
to use, copy, modify, merge, publish, distribute, sublicense, and/or sell 
copies of the Software, and to permit persons to whom the Software is 
furnished to do so, subject to the following conditions:

The above copyright notice and this permission notice shall be included in 
all copies or substantial portions of the Software.

THE SOFTWARE IS PROVIDED "AS IS", WITHOUT WARRANTY OF ANY KIND, EXPRESS OR 
IMPLIED, INCLUDING BUT NOT LIMITED TO THE WARRANTIES OF MERCHANTABILITY, 
FITNESS FOR A PARTICULAR PURPOSE AND NONINFRINGEMENT. IN NO EVENT SHALL THE 
AUTHORS OR COPYRIGHT HOLDERS BE LIABLE FOR ANY CLAIM, DAMAGES OR OTHER 
LIABILITY, WHETHER IN AN ACTION OF CONTRACT, TORT OR OTHERWISE, ARISING FROM, 
OUT OF OR IN CONNECTION WITH THE SOFTWARE OR THE USE OR OTHER DEALINGS 
IN THE SOFTWARE.
*)
// as long as VG is not at HR, it is going to HR
(*IF NOT(VG.state = VG_State.AT_HR) THEN
	VG.state := VG_State.FROM_DEFAULT_POS_TO_HR;
	vg_move_to_pos(x := 0, y := 0, z := 206);
	fin := vg_move_to_pos.fin;
	IF fin THEN
		VG.state := VG_State.AT_HR;
	END_IF
END_IF *)

VG.state := VG_State.AT_HR;
HR.state := HR_State.AT_CONVEYOR_BOX_FULL;
END_ACTION

ACTION ZBack_VG_TO_FU_active_active_0:
(*
Copyright (c) 2019 Manuel Goester, Michael Witt, Klaus Kammerer
Institute of Databases and Information Systems, Ulm University, Germany

Permission is hereby granted, free of charge, to any person obtaining a copy 
of this software and associated documentation files (the "Software"), to deal 
in the Software without restriction, including without limitation the rights 
to use, copy, modify, merge, publish, distribute, sublicense, and/or sell 
copies of the Software, and to permit persons to whom the Software is 
furnished to do so, subject to the following conditions:

The above copyright notice and this permission notice shall be included in 
all copies or substantial portions of the Software.

THE SOFTWARE IS PROVIDED "AS IS", WITHOUT WARRANTY OF ANY KIND, EXPRESS OR 
IMPLIED, INCLUDING BUT NOT LIMITED TO THE WARRANTIES OF MERCHANTABILITY, 
FITNESS FOR A PARTICULAR PURPOSE AND NONINFRINGEMENT. IN NO EVENT SHALL THE 
AUTHORS OR COPYRIGHT HOLDERS BE LIABLE FOR ANY CLAIM, DAMAGES OR OTHER 
LIABILITY, WHETHER IN AN ACTION OF CONTRACT, TORT OR OTHERWISE, ARISING FROM, 
OUT OF OR IN CONNECTION WITH THE SOFTWARE OR THE USE OR OTHER DEALINGS 
IN THE SOFTWARE.
*)
IF NOT(VG.sHorizontal) THEN
	VG.mHorizontalBackward := TRUE;
ELSE
	VG.mHorizontalBackward := FALSE;
	zFin := TRUE;
END_IF
END_ACTION

ACTION ZLeft_AND_XForward_VG_TO_FU_active_exit:
(*
Copyright (c) 2019 Manuel Goester, Michael Witt, Klaus Kammerer
Institute of Databases and Information Systems, Ulm University, Germany

Permission is hereby granted, free of charge, to any person obtaining a copy 
of this software and associated documentation files (the "Software"), to deal 
in the Software without restriction, including without limitation the rights 
to use, copy, modify, merge, publish, distribute, sublicense, and/or sell 
copies of the Software, and to permit persons to whom the Software is 
furnished to do so, subject to the following conditions:

The above copyright notice and this permission notice shall be included in 
all copies or substantial portions of the Software.

THE SOFTWARE IS PROVIDED "AS IS", WITHOUT WARRANTY OF ANY KIND, EXPRESS OR 
IMPLIED, INCLUDING BUT NOT LIMITED TO THE WARRANTIES OF MERCHANTABILITY, 
FITNESS FOR A PARTICULAR PURPOSE AND NONINFRINGEMENT. IN NO EVENT SHALL THE 
AUTHORS OR COPYRIGHT HOLDERS BE LIABLE FOR ANY CLAIM, DAMAGES OR OTHER 
LIABILITY, WHETHER IN AN ACTION OF CONTRACT, TORT OR OTHERWISE, ARISING FROM, 
OUT OF OR IN CONNECTION WITH THE SOFTWARE OR THE USE OR OTHER DEALINGS 
IN THE SOFTWARE.
*)
fin := FALSE;
END_ACTION

ACTION VG_WAIT_FOR_SL_active:
(*
Copyright (c) 2019 Manuel Goester, Michael Witt, Klaus Kammerer
Institute of Databases and Information Systems, Ulm University, Germany

Permission is hereby granted, free of charge, to any person obtaining a copy 
of this software and associated documentation files (the "Software"), to deal 
in the Software without restriction, including without limitation the rights 
to use, copy, modify, merge, publish, distribute, sublicense, and/or sell 
copies of the Software, and to permit persons to whom the Software is 
furnished to do so, subject to the following conditions:

The above copyright notice and this permission notice shall be included in 
all copies or substantial portions of the Software.

THE SOFTWARE IS PROVIDED "AS IS", WITHOUT WARRANTY OF ANY KIND, EXPRESS OR 
IMPLIED, INCLUDING BUT NOT LIMITED TO THE WARRANTIES OF MERCHANTABILITY, 
FITNESS FOR A PARTICULAR PURPOSE AND NONINFRINGEMENT. IN NO EVENT SHALL THE 
AUTHORS OR COPYRIGHT HOLDERS BE LIABLE FOR ANY CLAIM, DAMAGES OR OTHER 
LIABILITY, WHETHER IN AN ACTION OF CONTRACT, TORT OR OTHERWISE, ARISING FROM, 
OUT OF OR IN CONNECTION WITH THE SOFTWARE OR THE USE OR OTHER DEALINGS 
IN THE SOFTWARE.
*)
VG.state := VG_State.WAIT_FOR_SL;
END_ACTION

ACTION VG_WAIT_FOR_SL_exit:
(*
Copyright (c) 2019 Manuel Goester, Michael Witt, Klaus Kammerer
Institute of Databases and Information Systems, Ulm University, Germany

Permission is hereby granted, free of charge, to any person obtaining a copy 
of this software and associated documentation files (the "Software"), to deal 
in the Software without restriction, including without limitation the rights 
to use, copy, modify, merge, publish, distribute, sublicense, and/or sell 
copies of the Software, and to permit persons to whom the Software is 
furnished to do so, subject to the following conditions:

The above copyright notice and this permission notice shall be included in 
all copies or substantial portions of the Software.

THE SOFTWARE IS PROVIDED "AS IS", WITHOUT WARRANTY OF ANY KIND, EXPRESS OR 
IMPLIED, INCLUDING BUT NOT LIMITED TO THE WARRANTIES OF MERCHANTABILITY, 
FITNESS FOR A PARTICULAR PURPOSE AND NONINFRINGEMENT. IN NO EVENT SHALL THE 
AUTHORS OR COPYRIGHT HOLDERS BE LIABLE FOR ANY CLAIM, DAMAGES OR OTHER 
LIABILITY, WHETHER IN AN ACTION OF CONTRACT, TORT OR OTHERWISE, ARISING FROM, 
OUT OF OR IN CONNECTION WITH THE SOFTWARE OR THE USE OR OTHER DEALINGS 
IN THE SOFTWARE.
*)
fin := FALSE;
END_ACTION

ACTION VG_YUp_active:
(*
Copyright (c) 2019 Manuel Goester, Michael Witt, Klaus Kammerer
Institute of Databases and Information Systems, Ulm University, Germany

Permission is hereby granted, free of charge, to any person obtaining a copy 
of this software and associated documentation files (the "Software"), to deal 
in the Software without restriction, including without limitation the rights 
to use, copy, modify, merge, publish, distribute, sublicense, and/or sell 
copies of the Software, and to permit persons to whom the Software is 
furnished to do so, subject to the following conditions:

The above copyright notice and this permission notice shall be included in 
all copies or substantial portions of the Software.

THE SOFTWARE IS PROVIDED "AS IS", WITHOUT WARRANTY OF ANY KIND, EXPRESS OR 
IMPLIED, INCLUDING BUT NOT LIMITED TO THE WARRANTIES OF MERCHANTABILITY, 
FITNESS FOR A PARTICULAR PURPOSE AND NONINFRINGEMENT. IN NO EVENT SHALL THE 
AUTHORS OR COPYRIGHT HOLDERS BE LIABLE FOR ANY CLAIM, DAMAGES OR OTHER 
LIABILITY, WHETHER IN AN ACTION OF CONTRACT, TORT OR OTHERWISE, ARISING FROM, 
OUT OF OR IN CONNECTION WITH THE SOFTWARE OR THE USE OR OTHER DEALINGS 
IN THE SOFTWARE.
*)
IF NOT(VG.sVertical) THEN
	VG.mVerticalUp := TRUE;
ELSE
	VG.mVerticalUp := FALSE;
	VG.cY := 0;
	fin := TRUE;
END_IF
END_ACTION

ACTION VG_YUp_exit:
(*
Copyright (c) 2019 Manuel Goester, Michael Witt, Klaus Kammerer
Institute of Databases and Information Systems, Ulm University, Germany

Permission is hereby granted, free of charge, to any person obtaining a copy 
of this software and associated documentation files (the "Software"), to deal 
in the Software without restriction, including without limitation the rights 
to use, copy, modify, merge, publish, distribute, sublicense, and/or sell 
copies of the Software, and to permit persons to whom the Software is 
furnished to do so, subject to the following conditions:

The above copyright notice and this permission notice shall be included in 
all copies or substantial portions of the Software.

THE SOFTWARE IS PROVIDED "AS IS", WITHOUT WARRANTY OF ANY KIND, EXPRESS OR 
IMPLIED, INCLUDING BUT NOT LIMITED TO THE WARRANTIES OF MERCHANTABILITY, 
FITNESS FOR A PARTICULAR PURPOSE AND NONINFRINGEMENT. IN NO EVENT SHALL THE 
AUTHORS OR COPYRIGHT HOLDERS BE LIABLE FOR ANY CLAIM, DAMAGES OR OTHER 
LIABILITY, WHETHER IN AN ACTION OF CONTRACT, TORT OR OTHERWISE, ARISING FROM, 
OUT OF OR IN CONNECTION WITH THE SOFTWARE OR THE USE OR OTHER DEALINGS 
IN THE SOFTWARE.
*)
fin := FALSE;
END_ACTION

ACTION VG_TO_EJECT_POINT_exit:
(*
Copyright (c) 2019 Manuel Goester, Michael Witt, Klaus Kammerer
Institute of Databases and Information Systems, Ulm University, Germany

Permission is hereby granted, free of charge, to any person obtaining a copy 
of this software and associated documentation files (the "Software"), to deal 
in the Software without restriction, including without limitation the rights 
to use, copy, modify, merge, publish, distribute, sublicense, and/or sell 
copies of the Software, and to permit persons to whom the Software is 
furnished to do so, subject to the following conditions:

The above copyright notice and this permission notice shall be included in 
all copies or substantial portions of the Software.

THE SOFTWARE IS PROVIDED "AS IS", WITHOUT WARRANTY OF ANY KIND, EXPRESS OR 
IMPLIED, INCLUDING BUT NOT LIMITED TO THE WARRANTIES OF MERCHANTABILITY, 
FITNESS FOR A PARTICULAR PURPOSE AND NONINFRINGEMENT. IN NO EVENT SHALL THE 
AUTHORS OR COPYRIGHT HOLDERS BE LIABLE FOR ANY CLAIM, DAMAGES OR OTHER 
LIABILITY, WHETHER IN AN ACTION OF CONTRACT, TORT OR OTHERWISE, ARISING FROM, 
OUT OF OR IN CONNECTION WITH THE SOFTWARE OR THE USE OR OTHER DEALINGS 
IN THE SOFTWARE.
*)
fin := FALSE;
END_ACTION

ACTION VG_EJECT_active:
(*
Copyright (c) 2019 Manuel Goester, Michael Witt, Klaus Kammerer
Institute of Databases and Information Systems, Ulm University, Germany

Permission is hereby granted, free of charge, to any person obtaining a copy 
of this software and associated documentation files (the "Software"), to deal 
in the Software without restriction, including without limitation the rights 
to use, copy, modify, merge, publish, distribute, sublicense, and/or sell 
copies of the Software, and to permit persons to whom the Software is 
furnished to do so, subject to the following conditions:

The above copyright notice and this permission notice shall be included in 
all copies or substantial portions of the Software.

THE SOFTWARE IS PROVIDED "AS IS", WITHOUT WARRANTY OF ANY KIND, EXPRESS OR 
IMPLIED, INCLUDING BUT NOT LIMITED TO THE WARRANTIES OF MERCHANTABILITY, 
FITNESS FOR A PARTICULAR PURPOSE AND NONINFRINGEMENT. IN NO EVENT SHALL THE 
AUTHORS OR COPYRIGHT HOLDERS BE LIABLE FOR ANY CLAIM, DAMAGES OR OTHER 
LIABILITY, WHETHER IN AN ACTION OF CONTRACT, TORT OR OTHERWISE, ARISING FROM, 
OUT OF OR IN CONNECTION WITH THE SOFTWARE OR THE USE OR OTHER DEALINGS 
IN THE SOFTWARE.
*)
VG.valve := FALSE;
pneumatic_loaded := FALSE;
timer(IN:= TRUE, PT:= T#1S);
IF NOT(timer.Q = FALSE AND timer.IN) THEN
	// reset timer
	timer(IN:= FALSE);
	
	fin := TRUE;
END_IF
END_ACTION

ACTION VG_EJECT_exit:
(*
Copyright (c) 2019 Manuel Goester, Michael Witt, Klaus Kammerer
Institute of Databases and Information Systems, Ulm University, Germany

Permission is hereby granted, free of charge, to any person obtaining a copy 
of this software and associated documentation files (the "Software"), to deal 
in the Software without restriction, including without limitation the rights 
to use, copy, modify, merge, publish, distribute, sublicense, and/or sell 
copies of the Software, and to permit persons to whom the Software is 
furnished to do so, subject to the following conditions:

The above copyright notice and this permission notice shall be included in 
all copies or substantial portions of the Software.

THE SOFTWARE IS PROVIDED "AS IS", WITHOUT WARRANTY OF ANY KIND, EXPRESS OR 
IMPLIED, INCLUDING BUT NOT LIMITED TO THE WARRANTIES OF MERCHANTABILITY, 
FITNESS FOR A PARTICULAR PURPOSE AND NONINFRINGEMENT. IN NO EVENT SHALL THE 
AUTHORS OR COPYRIGHT HOLDERS BE LIABLE FOR ANY CLAIM, DAMAGES OR OTHER 
LIABILITY, WHETHER IN AN ACTION OF CONTRACT, TORT OR OTHERWISE, ARISING FROM, 
OUT OF OR IN CONNECTION WITH THE SOFTWARE OR THE USE OR OTHER DEALINGS 
IN THE SOFTWARE.
*)
fin := FALSE;
END_ACTION

ACTION BACK_TO_DEFAULT_active:
(*
Copyright (c) 2019 Manuel Goester, Michael Witt, Klaus Kammerer
Institute of Databases and Information Systems, Ulm University, Germany

Permission is hereby granted, free of charge, to any person obtaining a copy 
of this software and associated documentation files (the "Software"), to deal 
in the Software without restriction, including without limitation the rights 
to use, copy, modify, merge, publish, distribute, sublicense, and/or sell 
copies of the Software, and to permit persons to whom the Software is 
furnished to do so, subject to the following conditions:

The above copyright notice and this permission notice shall be included in 
all copies or substantial portions of the Software.

THE SOFTWARE IS PROVIDED "AS IS", WITHOUT WARRANTY OF ANY KIND, EXPRESS OR 
IMPLIED, INCLUDING BUT NOT LIMITED TO THE WARRANTIES OF MERCHANTABILITY, 
FITNESS FOR A PARTICULAR PURPOSE AND NONINFRINGEMENT. IN NO EVENT SHALL THE 
AUTHORS OR COPYRIGHT HOLDERS BE LIABLE FOR ANY CLAIM, DAMAGES OR OTHER 
LIABILITY, WHETHER IN AN ACTION OF CONTRACT, TORT OR OTHERWISE, ARISING FROM, 
OUT OF OR IN CONNECTION WITH THE SOFTWARE OR THE USE OR OTHER DEALINGS 
IN THE SOFTWARE.
*)
// Brings VG to its default pos where sVertical = sHorizontal = sRotation = 1
// 1. y-Axis 2. z-Axis 3. rotation
IF NOT(VG.sVertical) THEN
	VG.mVerticalUp := TRUE;
ELSE
	VG.mVerticalUp := FALSE;
	IF NOT(VG.sHorizontal) THEN
		VG.mHorizontalBackward := TRUE;
	ELSE
		VG.mHorizontalBackward := FALSE;
		IF NOT(VG.sRotation) THEN
			VG.mRotationClockwise := TRUE;
		ELSE
			VG.mRotationClockwise := FALSE;
			// default pos reached
			VG.state := VG_State.AT_DEFAULT_POS;
			VG.cX := 0;
			VG.cY := 0;
			VG.cZ := 0;
		END_IF
	END_IF
END_IF
END_ACTION

ACTION VG_TO_SL_exit:
(*
Copyright (c) 2019 Manuel Goester, Michael Witt, Klaus Kammerer
Institute of Databases and Information Systems, Ulm University, Germany

Permission is hereby granted, free of charge, to any person obtaining a copy 
of this software and associated documentation files (the "Software"), to deal 
in the Software without restriction, including without limitation the rights 
to use, copy, modify, merge, publish, distribute, sublicense, and/or sell 
copies of the Software, and to permit persons to whom the Software is 
furnished to do so, subject to the following conditions:

The above copyright notice and this permission notice shall be included in 
all copies or substantial portions of the Software.

THE SOFTWARE IS PROVIDED "AS IS", WITHOUT WARRANTY OF ANY KIND, EXPRESS OR 
IMPLIED, INCLUDING BUT NOT LIMITED TO THE WARRANTIES OF MERCHANTABILITY, 
FITNESS FOR A PARTICULAR PURPOSE AND NONINFRINGEMENT. IN NO EVENT SHALL THE 
AUTHORS OR COPYRIGHT HOLDERS BE LIABLE FOR ANY CLAIM, DAMAGES OR OTHER 
LIABILITY, WHETHER IN AN ACTION OF CONTRACT, TORT OR OTHERWISE, ARISING FROM, 
OUT OF OR IN CONNECTION WITH THE SOFTWARE OR THE USE OR OTHER DEALINGS 
IN THE SOFTWARE.
*)
step := 1;
END_ACTION

ACTION VG_DIRECTLY_EJECT_W_active:
(*
Copyright (c) 2019 Manuel Goester, Michael Witt, Klaus Kammerer
Institute of Databases and Information Systems, Ulm University, Germany

Permission is hereby granted, free of charge, to any person obtaining a copy 
of this software and associated documentation files (the "Software"), to deal 
in the Software without restriction, including without limitation the rights 
to use, copy, modify, merge, publish, distribute, sublicense, and/or sell 
copies of the Software, and to permit persons to whom the Software is 
furnished to do so, subject to the following conditions:

The above copyright notice and this permission notice shall be included in 
all copies or substantial portions of the Software.

THE SOFTWARE IS PROVIDED "AS IS", WITHOUT WARRANTY OF ANY KIND, EXPRESS OR 
IMPLIED, INCLUDING BUT NOT LIMITED TO THE WARRANTIES OF MERCHANTABILITY, 
FITNESS FOR A PARTICULAR PURPOSE AND NONINFRINGEMENT. IN NO EVENT SHALL THE 
AUTHORS OR COPYRIGHT HOLDERS BE LIABLE FOR ANY CLAIM, DAMAGES OR OTHER 
LIABILITY, WHETHER IN AN ACTION OF CONTRACT, TORT OR OTHERWISE, ARISING FROM, 
OUT OF OR IN CONNECTION WITH THE SOFTWARE OR THE USE OR OTHER DEALINGS 
IN THE SOFTWARE.
*)
CASE step OF
	1:
		// z axis: from HR to EJECT
		// decide to which eject point to go by color
		IF NOT(fin) THEN
			IF TC.batchJobQueue.batchJobs[TC.currBatchJobIdx].workpieces[TC.batchJobQueue.batchJobs[TC.currBatchJobIdx].nextNotProcessedIdx].color = 'white' THEN
				// go to eject point 1
				vg_move_to_pos(x := 0, y := 0, z := 2);
			ELSIF TC.batchJobQueue.batchJobs[TC.currBatchJobIdx].workpieces[TC.batchJobQueue.batchJobs[TC.currBatchJobIdx].nextNotProcessedIdx].color = 'red' THEN
				// go to eject point 2
				vg_move_to_pos(x := 0, y := 0, z := 15);
			ELSIF TC.batchJobQueue.batchJobs[TC.currBatchJobIdx].workpieces[TC.batchJobQueue.batchJobs[TC.currBatchJobIdx].nextNotProcessedIdx].color = 'blue' THEN
				// go to eject point 3
				vg_move_to_pos(x := 0, y := 0, z := 23);
			ELSE
				// if color is unknown, go to eject point 1
				vg_move_to_pos(x := 0, y := 0, z := 2);
			END_IF
			fin := vg_move_to_pos.fin;
		ELSE
			fin := FALSE;
			step := step + 1;
		END_IF
	2:
		// x and y axis: go to eject point
		IF NOT(fin) THEN
			IF TC.batchJobQueue.batchJobs[TC.currBatchJobIdx].workpieces[TC.batchJobQueue.batchJobs[TC.currBatchJobIdx].nextNotProcessedIdx].color = 'white' THEN
				// go to eject point 1
				vg_move_to_pos(x := 25, y := 133, z := 2);
				VG.state := VG_State.AT_EJECT_1;
			ELSIF TC.batchJobQueue.batchJobs[TC.currBatchJobIdx].workpieces[TC.batchJobQueue.batchJobs[TC.currBatchJobIdx].nextNotProcessedIdx].color = 'red' THEN
				// go to eject point 2
				vg_move_to_pos(x := 30, y := 133, z := 15);
				VG.state := VG_State.AT_EJECT_2;
			ELSIF TC.batchJobQueue.batchJobs[TC.currBatchJobIdx].workpieces[TC.batchJobQueue.batchJobs[TC.currBatchJobIdx].nextNotProcessedIdx].color = 'blue' THEN
				// go to eject point 3
				vg_move_to_pos(x := 49, y := 133, z := 23);
				VG.state := VG_State.AT_EJECT_3;
			ELSE
				// if color is unknown, go to eject point 1
				vg_move_to_pos(x := 25, y := 133, z := 2);
				VG.state := VG_State.AT_EJECT_1;
			END_IF
			fin := vg_move_to_pos.fin;
		ELSE
			fin := FALSE;
			step := step + 1;
		END_IF
	3:
		// open valve to drop workpiece
		VG.valve := FALSE;
		pneumatic_loaded := FALSE;
		timer(IN:= TRUE, PT:= T#1S);
		IF NOT(timer.Q = FALSE AND timer.IN) THEN
			// reset timer
			timer(IN:= FALSE);
			step := step + 1;
		END_IF
	4:
		// Brings VG to its default pos
		IF NOT(VG.sVertical) THEN
			VG.mVerticalUp := TRUE;
		ELSE
			VG.mVerticalUp := FALSE;
			VG.cY := 0;
		END_IF
		IF NOT(VG.sHorizontal) THEN
			VG.mHorizontalBackward := TRUE;
		ELSE
			VG.mHorizontalBackward := FALSE;
			VG.cX := 0;
		END_IF
		IF NOT(VG.sRotation) THEN
			VG.mRotationClockwise := TRUE;
		ELSE
			VG.mRotationClockwise := FALSE;
			VG.cZ := 0;
		END_IF
		
		IF VG.sHorizontal AND VG.sVertical AND VG.sRotation THEN
			// default pos reached
			VG.state := VG_State.AT_DEFAULT_POS;
			// finished
			step := 1;
		END_IF
END_CASE
END_ACTION

ACTION VG_TO_HR_exit:
(*
Copyright (c) 2019 Manuel Goester, Michael Witt, Klaus Kammerer
Institute of Databases and Information Systems, Ulm University, Germany

Permission is hereby granted, free of charge, to any person obtaining a copy 
of this software and associated documentation files (the "Software"), to deal 
in the Software without restriction, including without limitation the rights 
to use, copy, modify, merge, publish, distribute, sublicense, and/or sell 
copies of the Software, and to permit persons to whom the Software is 
furnished to do so, subject to the following conditions:

The above copyright notice and this permission notice shall be included in 
all copies or substantial portions of the Software.

THE SOFTWARE IS PROVIDED "AS IS", WITHOUT WARRANTY OF ANY KIND, EXPRESS OR 
IMPLIED, INCLUDING BUT NOT LIMITED TO THE WARRANTIES OF MERCHANTABILITY, 
FITNESS FOR A PARTICULAR PURPOSE AND NONINFRINGEMENT. IN NO EVENT SHALL THE 
AUTHORS OR COPYRIGHT HOLDERS BE LIABLE FOR ANY CLAIM, DAMAGES OR OTHER 
LIABILITY, WHETHER IN AN ACTION OF CONTRACT, TORT OR OTHERWISE, ARISING FROM, 
OUT OF OR IN CONNECTION WITH THE SOFTWARE OR THE USE OR OTHER DEALINGS 
IN THE SOFTWARE.
*)
fin := FALSE;
END_ACTION

END_PROGRAM

// Device/Application/VG/FBs/VG_MOVE
(*
	Moves VG in x, y and z axis
	
Copyright (c) 2019 Manuel Goester, Michael Witt, Klaus Kammerer
Institute of Databases and Information Systems, Ulm University, Germany

Permission is hereby granted, free of charge, to any person obtaining a copy 
of this software and associated documentation files (the "Software"), to deal 
in the Software without restriction, including without limitation the rights 
to use, copy, modify, merge, publish, distribute, sublicense, and/or sell 
copies of the Software, and to permit persons to whom the Software is 
furnished to do so, subject to the following conditions:

The above copyright notice and this permission notice shall be included in 
all copies or substantial portions of the Software.

THE SOFTWARE IS PROVIDED "AS IS", WITHOUT WARRANTY OF ANY KIND, EXPRESS OR 
IMPLIED, INCLUDING BUT NOT LIMITED TO THE WARRANTIES OF MERCHANTABILITY, 
FITNESS FOR A PARTICULAR PURPOSE AND NONINFRINGEMENT. IN NO EVENT SHALL THE 
AUTHORS OR COPYRIGHT HOLDERS BE LIABLE FOR ANY CLAIM, DAMAGES OR OTHER 
LIABILITY, WHETHER IN AN ACTION OF CONTRACT, TORT OR OTHERWISE, ARISING FROM, 
OUT OF OR IN CONNECTION WITH THE SOFTWARE OR THE USE OR OTHER DEALINGS 
IN THE SOFTWARE.
*)
FUNCTION_BLOCK VG_MOVE
VAR_INPUT
	// distance VG will go forward (positive value) or backward (negative value)
	x: INT;
	/// distance VG will go down (positive value) or up (negative value)
	y: INT;
	// distance VG will go counter clockwise (positive value) or clockwise (negative value)
	z: INT;
END_VAR
VAR_OUTPUT
	
END_VAR
VAR	
	// finish flags
	xFin: BOOL := FALSE;
	yFin: BOOL := FALSE;
	zFin: BOOL := FALSE;
	fin: BOOL := FALSE;
	// true, if an impulse coming from the motor has been already counted
	xAlreadyCounted: BOOL := FALSE;
	yAlreadyCounted: BOOL := FALSE;
	zAlreadyCounted: BOOL := FALSE;
	// counters
	cX: INT := 0;
	cY: INT := 0;
	cZ: INT := 0;
END_VAR

fin := FALSE;

// X AXIS (Forward/Backward)
IF x < 0 THEN
	// drive backward
	IF cX = x THEN
		// if counter reached demanded position, we're done
		VG.mHorizontalBackward := FALSE;
		xFin := TRUE;
	ELSE
		xFin := FALSE;
		IF cX > x THEN
			VG.mHorizontalBackward := TRUE;
			IF VG.encHorizontal AND NOT(xAlreadyCounted) THEN
				// update local counter
				cX := cX - 1;
				// update global counter
				VG.cX := VG.cX - 1;
				xAlreadyCounted := TRUE;
			ELSIF NOT(VG.encHorizontal) THEN
				xAlreadyCounted := FALSE;
			END_IF
		END_IF
	END_IF
ELSE
	// x >= 0
	// drive forward
	IF cX = x THEN
		// if counter reached demanded position, we're done
		VG.mHorizontalForward := FALSE;
		xFin := TRUE;
	ELSE
		xFin := FALSE;
		IF cX < x THEN
			VG.mHorizontalForward := TRUE;
			IF VG.encHorizontal AND NOT(xAlreadyCounted) THEN
				// update local counter
				cX := cX + 1;
				// update global counter
				VG.cX := VG.cX + 1;
				xAlreadyCounted := TRUE;
			ELSIF NOT(VG.encHorizontal) THEN
				xAlreadyCounted := FALSE;
			END_IF
		END_IF
	END_IF
END_IF

// Y AXIS (Up/Down)
IF y < 0 THEN
	// drive up
	IF cY = y THEN
		// if counter reached demanded position, we're done
		VG.mVerticalUp := FALSE;
		yFin := TRUE;
	ELSE
		yFin := FALSE;
		IF cY > y THEN
			VG.mVerticalUp := TRUE;
			IF VG.encVertical AND NOT(yAlreadyCounted) THEN
				// update local counter
				cY := cY - 1;
				// update global counter
				VG.cY := VG.cY - 1;
				yAlreadyCounted := TRUE;
			ELSIF NOT(VG.encVertical) THEN
				yAlreadyCounted := FALSE;
			END_IF
		END_IF
	END_IF
ELSE
	// y >= 0
	// drive down
	IF cY = y THEN
		// if counter reached demanded position, we're done
		VG.mVerticalDown := FALSE;
	yFin := TRUE;
	ELSE
		yFin := FALSE;
		IF cY < y THEN
			VG.mVerticalDown := TRUE;
			IF VG.encVertical AND NOT(yAlreadyCounted) THEN
				// update local counter
				cY := cY + 1;
				// update global counter
				VG.cY := VG.cY + 1;
				yAlreadyCounted := TRUE;
			ELSIF NOT(VG.encVertical) THEN
				yAlreadyCounted := FALSE;
			END_IF
		END_IF
	END_IF
END_IF

// Z AXIS (Rotation)
IF z < 0 THEN
	// drive clockwise
	IF cZ = z THEN
		// if counter reached demanded position, we're done
		VG.mRotationClockwise := FALSE;
		zFin := TRUE;
	ELSE
		zFin := FALSE;
		IF cZ > z THEN
			VG.mRotationClockwise := TRUE;
			IF VG.encRotation AND NOT(zAlreadyCounted) THEN
				// update local counter
				cZ := cZ - 1;
				// update global counter
				VG.cZ := VG.cZ - 1;
				zAlreadyCounted := TRUE;
			ELSIF NOT(VG.encRotation) THEN
				zAlreadyCounted := FALSE;
			END_IF
		END_IF
	END_IF
ELSE
	// z >= 0
	// drive counter clockwise
	IF cZ = z THEN
		// if counter reached demanded position, we're done
		VG.mRotationCClockwise := FALSE;
		zFin := TRUE;
	ELSE
		zFin := FALSE;
		IF cZ < z THEN
			VG.mRotationCClockwise := TRUE;
			IF VG.encRotation AND NOT(zAlreadyCounted) THEN
				// update local counter
				cZ := cZ + 1;
				// update global counter
				VG.cZ := VG.cZ + 1;
				zAlreadyCounted := TRUE;
			ELSIF NOT(VG.encRotation) THEN
				zAlreadyCounted := FALSE;
			END_IF
		END_IF
	END_IF
END_IF

